  MoveL 627 to (56, 272.86, 210) mm, rotated rx -72.12 ry -13.76 rz 133.16 deg; joints [-11.184, -48.256, 111.238, -158.714, 116.997, -159.582, -1249.582]
  MoveL 628 to (57.57, 267.12, 200) mm, rotated rx -73 ry -11.66 rz 121.38 deg; joints [-11.86, -51.281, 112.071, -161.907, 109.412, -163.121, -1243.4]
  MoveL 629 to (58.59, 260.98, 190) mm, rotated rx -71.71 ry -12.29 rz 118.09 deg; joints [-12.413, -49.73, 111.982, -161.392, 113.738, -160.153, -1237.009]
  MoveL 630 to (58.95, 254.55, 180) mm, rotated rx -70.55 ry -13.02 rz 114.47 deg; joints [-12.913, -48.175, 111.692, -160.589, 117.696, -157.241, -1230.447]
  MoveL 631 to (58.59, 247.92, 170) mm, rotated rx -71.88 ry -10.84 rz 101.84 deg; joints [-13.52, -51.449, 112.574, -163.918, 109.603, -161.344, -1223.752]
  MoveL 632 to (57.45, 241.22, 160) mm, rotated rx -70.86 ry -11.6 rz 97.82 deg; joints [-13.978, -50.056, 112.473, -163.221, 113.479, -158.849, -1216.959]
  MoveL 633 to (55.51, 234.59, 150) mm, rotated rx -69.95 ry -12.44 rz 93.68 deg; joints [-14.39, -48.623, 112.206, -162.264, 117.149, -156.334, -1210.107]
  MoveL 634 to (52.77, 228.15, 140) mm, rotated rx -71.59 ry -10.32 rz 80.79 deg; joints [-14.925, -51.956, 113.016, -165.486, 108.844, -160.666, -1203.231]
  MoveL 635 to (49.26, 222.05, 130) mm, rotated rx -70.76 ry -11.22 rz 76.66 deg; joints [-15.304, -50.588, 112.931, -164.581, 112.697, -158.413, -1196.367]
  MoveL 636 to (45.04, 216.4, 120) mm, rotated rx -70.03 ry -12.23 rz 72.63 deg; joints [-15.637, -49.129, 112.673, -163.392, 116.478, -156.06, -1189.55]
  MoveL 637 to (40.19, 211.31, 110) mm, rotated rx -71.83 ry -10.32 rz 60.03 deg; joints [-16.092, -52.366, 113.385, -166.332, 108.333, -160.403, -1182.816]
  MoveL 638 to (34.83, 206.87, 100) mm, rotated rx -71.13 ry -11.44 rz 56.41 deg; joints [-16.388, -50.868, 113.282, -165.098, 112.545, -158.165, -1176.2]
  MoveL 639 to (29.06, 203.14, 90) mm, rotated rx -70.54 ry -12.69 rz 53.09 deg; joints [-16.632, -49.217, 112.963, -163.507, 116.784, -155.729, -1169.736]
  MoveL 640 to (23.03, 200.17, 80) mm, rotated rx -72.37 ry -11.13 rz 41.37 deg; joints [-17.001, -52.244, 113.649, -166.075, 109.258, -159.979, -1163.458]
  MoveL 641 to (16.86, 197.94, 70) mm, rotated rx -71.8 ry -12.55 rz 38.86 deg; joints [-17.193, -50.441, 113.427, -164.304, 114.153, -157.511, -1157.4]
  MoveL 642 to (10.69, 196.46, 60) mm, rotated rx -73.66 ry -11.39 rz 28.02 deg; joints [-17.464, -53.158, 113.849, -166.257, 107.044, -161.446, -1151.595]
  MoveL 643 to (4.64, 195.67, 50) mm, rotated rx -73.16 ry -13.02 rz 26.6 deg; joints [-17.59, -51.134, 113.679, -164.198, 112.728, -158.838, -1146.075]
  MoveL 644 to (-1.18, 195.49, 40) mm, rotated rx -72.85 ry -14.8 rz 25.84 deg; joints [-17.639, -48.817, 113.11, -161.546, 118.515, -155.811, -1140.872]
  MoveL 645 to (-6.67, 195.86, 30) mm, rotated rx -74.62 ry -14.16 rz 16.83 deg; joints [-17.801, -51.19, 113.743, -163.089, 112.896, -159.64, -1136.017]
  MoveL 646 to (-11.76, 196.67, 20) mm, rotated rx -76.4 ry -13.89 rz 8.51 deg; joints [-17.869, -53.24, 113.964, -163.907, 107.44, -163.077, -1131.54]
  MoveL 647 to (-16.38, 197.8, 10) mm, rotated rx -78.17 ry -13.98 rz 0.96 deg; joints [-17.851, -54.956, 113.848, -164.09, 102.301, -166.234, -1127.469]
  MoveL 648 to (-20.49, 199.16, 0) mm, rotated rx -78.17 ry -13.98 rz 0.96 deg; joints [-18.269, -54.883, 113.526, -164.417, 102.002, -166.09, -1127.469]
  Set speed (1000.0 mm/s)
  MoveL 649 to (-20.49, 199.16, 0) mm, rotated rx -78.17 ry -13.98 rz 0.96 deg; joints [-18.269, -54.883, 113.526, -164.417, 102.002, -166.09, -1127.469]
  Set speed (1000.0 mm/s)
  MoveL 650 to (37.11, 300.24, 290) mm, rotated rx -90 ry -25 rz 177.31 deg; joints [-2.318, -51.586, 102.108, -141.879, 96.357, -189.349, -1307.315]
  MoveL 651 to (37.11, 300.24, 290) mm, rotated rx -90 ry -25 rz -172.69 deg; joints [-2.265, -48.205, 103.066, -142.213, 108.813, -182.608, -1307.315]
  Set speed (60.0 mm/s)
  MoveL 652 to (43.85, 319.91, 290) mm, rotated rx -90 ry -25 rz -166.2 deg; joints [-2.265, -49.125, 102.977, -142.419, 108.014, -183.258, -1313.803]
  Set speed (1000.0 mm/s)
  MoveL 653 to (43.85, 319.91, 290) mm, rotated rx -90 ry -25 rz -166.2 deg; joints [-2.265, -49.125, 102.977, -142.419, 108.014, -183.258, -1313.803]
  Set speed (1000.0 mm/s)
  MoveL 654 to (-20.49, 199.16, 0) mm, rotated rx -90 ry -25 rz 31.39 deg; joints [-13.282, -51.572, 108.683, -149.29, 107.197, -175.931, -1151.385]
  MoveL 655 to (-20.49, 199.16, 0) mm, rotated rx -90 ry -25 rz 31.39 deg; joints [-13.282, -51.572, 108.683, -149.29, 107.197, -175.931, -1151.385]
  Set speed (60.0 mm/s)
  MoveL 656 to (-20.57, 178.36, 0) mm, rotated rx -90 ry -25 rz 45.86 deg; joints [-13.325, -48.191, 107.994, -147.492, 118.47, -169.661, -1155.856]
  Set speed (1000.0 mm/s)
  MoveL 657 to (-20.57, 178.36, 0) mm, rotated rx -90 ry -25 rz 45.86 deg; joints [-13.325, -48.191, 107.994, -147.492, 118.47, -169.661, -1155.856]
  Set speed (1000.0 mm/s)
  MoveL 658 to (-20.49, 199.16, 0) mm, rotated rx -90 ry -25 rz 31.39 deg; joints [-13.282, -51.572, 108.683, -149.29, 107.197, -175.931, -1151.385]
  MoveL 659 to (-20.49, 199.16, 0) mm, rotated rx -90 ry -25 rz 31.39 deg; joints [-13.282, -51.572, 108.683, -149.29, 107.197, -175.931, -1151.385]
  Set speed (60.0 mm/s)
  MoveL 660 to (-16.38, 197.8, 10) mm, rotated rx -90 ry -25 rz 35.25 deg; joints [-12.889, -51.522, 108.574, -149.026, 107.257, -176.155, -1155.247]
  MoveL 661 to (-11.76, 196.67, 20) mm, rotated rx -90 ry -25 rz 39.48 deg; joints [-12.496, -51.468, 108.459, -148.763, 107.315, -176.379, -1159.483]
  MoveL 662 to (-6.67, 195.86, 30) mm, rotated rx -90 ry -25 rz 44.06 deg; joints [-12.104, -51.409, 108.339, -148.502, 107.374, -176.604, -1164.062]
  MoveL 663 to (-1.18, 195.49, 40) mm, rotated rx -90 ry -25 rz 48.95 deg; joints [-11.713, -51.345, 108.212, -148.241, 107.432, -176.829, -1168.952]
  MoveL 664 to (4.64, 195.67, 50) mm, rotated rx -90 ry -25 rz 54.12 deg; joints [-11.323, -51.276, 108.079, -147.982, 107.491, -177.054, -1174.124]
  MoveL 665 to (10.69, 196.46, 60) mm, rotated rx -90 ry -25 rz 59.55 deg; joints [-10.933, -51.201, 107.94, -147.724, 107.551, -177.279, -1179.549]
  MoveL 666 to (16.86, 197.94, 70) mm, rotated rx -90 ry -25 rz 65.2 deg; joints [-10.544, -51.119, 107.796, -147.467, 107.612, -177.504, -1185.201]
  MoveL 667 to (23.03, 200.17, 80) mm, rotated rx -90 ry -25 rz 71.05 deg; joints [-10.156, -51.031, 107.645, -147.21, 107.675, -177.728, -1191.051]
  MoveL 668 to (29.06, 203.14, 90) mm, rotated rx -90 ry -25 rz 77.07 deg; joints [-9.769, -50.937, 107.489, -146.955, 107.738, -177.951, -1197.074]
  MoveL 669 to (34.83, 206.87, 100) mm, rotated rx -90 ry -25 rz 83.24 deg; joints [-9.383, -50.836, 107.326, -146.701, 107.803, -178.174, -1203.245]
  MoveL 670 to (40.19, 211.31, 110) mm, rotated rx -90 ry -25 rz 89.54 deg; joints [-8.998, -50.729, 107.158, -146.448, 107.869, -178.396, -1209.537]
  MoveL 671 to (45.04, 216.4, 120) mm, rotated rx -90 ry -25 rz 95.93 deg; joints [-8.614, -50.616, 106.984, -146.196, 107.936, -178.617, -1215.926]
  MoveL 672 to (49.26, 222.05, 130) mm, rotated rx -90 ry -25 rz 102.38 deg; joints [-8.231, -50.497, 106.804, -145.946, 108.004, -178.839, -1222.384]
  MoveL 673 to (52.77, 228.15, 140) mm, rotated rx -90 ry -25 rz 108.88 deg; joints [-7.849, -50.373, 106.617, -145.697, 108.072, -179.06, -1228.885]
  MoveL 674 to (55.51, 234.59, 150) mm, rotated rx -90 ry -25 rz 115.4 deg; joints [-7.468, -50.244, 106.425, -145.449, 108.139, -179.281, -1235.4]
  MoveL 675 to (57.45, 241.22, 160) mm, rotated rx -90 ry -25 rz 121.9 deg; joints [-7.088, -50.111, 106.226, -145.203, 108.206, -179.504, -1241.898]
  MoveL 676 to (58.59, 247.92, 170) mm, rotated rx -90 ry -25 rz 128.35 deg; joints [-6.709, -49.974, 106.022, -144.958, 108.271, -179.727, -1248.348]
  MoveL 677 to (58.95, 254.55, 180) mm, rotated rx -90 ry -25 rz 134.71 deg; joints [-6.332, -49.834, 105.811, -144.716, 108.334, -179.952, -1254.714]
  MoveL 678 to (58.59, 260.98, 190) mm, rotated rx -90 ry -25 rz 140.96 deg; joints [-5.956, -49.691, 105.593, -144.476, 108.396, -180.178, -1260.96]
  MoveL 679 to (57.57, 267.12, 200) mm, rotated rx -90 ry -25 rz 147.05 deg; joints [-5.581, -49.547, 105.37, -144.238, 108.454, -180.407, -1267.046]
  MoveL 680 to (56, 272.86, 210) mm, rotated rx -90 ry -25 rz 152.93 deg; joints [-5.207, -49.401, 105.139, -144.002, 108.509, -180.639, -1272.931]
  MoveL 681 to (53.98, 278.14, 220) mm, rotated rx -90 ry -25 rz 158.57 deg; joints [-4.834, -49.254, 104.903, -143.769, 108.56, -180.873, -1278.571]
  MoveL 682 to (51.62, 282.9, 230) mm, rotated rx -90 ry -25 rz 163.92 deg; joints [-4.463, -49.106, 104.66, -143.538, 108.608, -181.111, -1283.922]
  MoveL 683 to (49.06, 287.12, 240) mm, rotated rx -90 ry -25 rz 168.94 deg; joints [-4.093, -48.957, 104.41, -143.31, 108.652, -181.352, -1288.935]
  MoveL 684 to (46.4, 290.79, 250) mm, rotated rx -90 ry -25 rz 173.57 deg; joints [-3.725, -48.808, 104.155, -143.085, 108.692, -181.596, -1293.565]
  MoveL 685 to (43.78, 293.91, 260) mm, rotated rx -90 ry -25 rz 177.77 deg; joints [-3.358, -48.659, 103.892, -142.863, 108.728, -181.844, -1297.765]
  MoveL 686 to (41.29, 296.51, 270) mm, rotated rx -90 ry -25 rz -178.51 deg; joints [-2.992, -48.508, 103.623, -142.644, 108.76, -182.095, -1301.487]
  MoveL 687 to (39.03, 298.61, 280) mm, rotated rx -90 ry -25 rz -175.31 deg; joints [-2.628, -48.357, 103.348, -142.427, 108.788, -182.35, -1304.686]
  MoveL 688 to (37.11, 300.24, 290) mm, rotated rx -90 ry -25 rz -172.69 deg; joints [-2.265, -48.205, 103.066, -142.213, 108.813, -182.608, -1307.315]
  Set speed (1000.0 mm/s)
  MoveL 689 to (37.11, 300.24, 290) mm, rotated rx -90 ry -25 rz -172.69 deg; joints [-2.265, -48.205, 103.066, -142.213, 108.813, -182.608, -1307.315]
  Set speed (1000.0 mm/s)
  MoveL 690 to (43.85, 319.91, 290) mm, rotated rx -90 ry -25 rz -166.2 deg; joints [-2.265, -49.125, 102.977, -142.419, 108.014, -183.258, -1313.803]
  MoveL 691 to (43.85, 319.91, 290) mm, rotated rx -90 ry -25 rz -166.2 deg; joints [-2.265, -49.125, 102.977, -142.419, 108.014, -183.258, -1313.803]
  Set speed (60.0 mm/s)
  MoveL 692 to (46.6, 317.98, 280) mm, rotated rx -90 ry -25 rz -168.79 deg; joints [-2.628, -49.278, 103.258, -142.631, 107.986, -182.998, -1311.207]
  MoveL 693 to (49.86, 315.46, 270) mm, rotated rx -90 ry -25 rz -171.95 deg; joints [-2.992, -49.431, 103.534, -142.847, 107.954, -182.741, -1308.046]
  MoveL 694 to (53.49, 312.31, 260) mm, rotated rx -90 ry -25 rz -175.64 deg; joints [-3.358, -49.582, 103.802, -143.065, 107.919, -182.487, -1304.36]
  MoveL 695 to (57.36, 308.47, 250) mm, rotated rx -90 ry -25 rz -179.81 deg; joints [-3.725, -49.733, 104.064, -143.286, 107.88, -182.237, -1300.194]
  MoveL 696 to (61.34, 303.9, 240) mm, rotated rx -90 ry -25 rz 175.59 deg; joints [-4.093, -49.883, 104.32, -143.51, 107.836, -181.989, -1295.591]
  MoveL 697 to (65.27, 298.59, 230) mm, rotated rx -90 ry -25 rz 170.6 deg; joints [-4.463, -50.032, 104.569, -143.736, 107.789, -181.746, -1290.596]
  MoveL 698 to (68.98, 292.54, 220) mm, rotated rx -90 ry -25 rz 165.25 deg; joints [-4.834, -50.18, 104.811, -143.966, 107.738, -181.505, -1285.253]
  MoveL 699 to (72.31, 285.76, 210) mm, rotated rx -90 ry -25 rz 159.61 deg; joints [-5.207, -50.328, 105.047, -144.197, 107.683, -181.268, -1279.605]
  MoveL 700 to (75.1, 278.3, 200) mm, rotated rx -90 ry -25 rz 153.7 deg; joints [-5.581, -50.475, 105.276, -144.432, 107.624, -181.034, -1273.697]
  MoveL 701 to (77.2, 270.26, 190) mm, rotated rx -90 ry -25 rz 147.57 deg; joints [-5.956, -50.621, 105.499, -144.668, 107.562, -180.802, -1267.571]
  MoveL 702 to (78.47, 261.74, 180) mm, rotated rx -90 ry -25 rz 141.27 deg; joints [-6.332, -50.765, 105.715, -144.907, 107.496, -180.573, -1261.269]
  MoveL 703 to (78.79, 252.87, 170) mm, rotated rx -90 ry -25 rz 134.83 deg; joints [-6.709, -50.906, 105.925, -145.148, 107.428, -180.346, -1254.829]
  MoveL 704 to (78.09, 243.82, 160) mm, rotated rx -90 ry -25 rz 128.29 deg; joints [-7.088, -51.045, 106.129, -145.391, 107.357, -180.121, -1248.29]
  MoveL 705 to (76.31, 234.75, 150) mm, rotated rx -90 ry -25 rz 121.69 deg; joints [-7.468, -51.181, 106.326, -145.636, 107.285, -179.896, -1241.689]
  MoveL 706 to (73.44, 225.85, 140) mm, rotated rx -90 ry -25 rz 115.06 deg; joints [-7.849, -51.313, 106.518, -145.882, 107.212, -179.673, -1235.058]
  MoveL 707 to (69.5, 217.29, 130) mm, rotated rx -90 ry -25 rz 108.43 deg; joints [-8.231, -51.44, 106.703, -146.13, 107.138, -179.45, -1228.432]
  MoveL 708 to (64.57, 209.26, 120) mm, rotated rx -90 ry -25 rz 101.84 deg; joints [-8.614, -51.562, 106.882, -146.38, 107.064, -179.227, -1221.84]
  MoveL 709 to (58.74, 201.9, 110) mm, rotated rx -90 ry -25 rz 95.31 deg; joints [-8.998, -51.679, 107.055, -146.63, 106.991, -179.004, -1215.313]
  MoveL 710 to (52.14, 195.34, 100) mm, rotated rx -90 ry -25 rz 88.88 deg; joints [-9.383, -51.79, 107.223, -146.882, 106.918, -178.781, -1208.879]
  MoveL 711 to (44.91, 189.68, 90) mm, rotated rx -90 ry -25 rz 92.57 deg; joints [-9.833, -47.57, 106.798, -145.465, 118.969, -171.706, -1202.567]
  MoveL 712 to (37.24, 184.98, 80) mm, rotated rx -90 ry -25 rz 86.4 deg; joints [-10.217, -47.663, 106.955, -145.686, 118.911, -171.479, -1196.403]
  MoveL 713 to (29.3, 181.28, 70) mm, rotated rx -90 ry -25 rz 80.42 deg; joints [-10.603, -47.75, 107.107, -145.908, 118.855, -171.251, -1190.416]
  MoveL 714 to (21.27, 178.55, 60) mm, rotated rx -90 ry -25 rz 74.63 deg; joints [-10.989, -47.83, 107.252, -146.131, 118.799, -171.024, -1184.633]
  MoveL 715 to (13.31, 176.76, 50) mm, rotated rx -90 ry -25 rz 69.08 deg; joints [-11.377, -47.903, 107.391, -146.354, 118.744, -170.796, -1179.083]
  MoveL 716 to (5.58, 175.83, 40) mm, rotated rx -90 ry -25 rz 63.79 deg; joints [-11.765, -47.971, 107.524, -146.579, 118.689, -170.567, -1173.794]
  MoveL 717 to (-1.77, 175.65, 30) mm, rotated rx -90 ry -25 rz 58.8 deg; joints [-12.154, -48.034, 107.651, -146.805, 118.635, -170.34, -1168.796]
  MoveL 718 to (-8.64, 176.1, 20) mm, rotated rx -90 ry -25 rz 54.12 deg; joints [-12.543, -48.091, 107.771, -147.033, 118.58, -170.112, -1164.119]
  MoveL 719 to (-14.93, 177.06, 10) mm, rotated rx -90 ry -25 rz 49.79 deg; joints [-12.934, -48.143, 107.885, -147.261, 118.526, -169.886, -1159.795]
  MoveL 720 to (-20.57, 178.36, 0) mm, rotated rx -90 ry -25 rz 45.86 deg; joints [-13.325, -48.191, 107.994, -147.492, 118.47, -169.661, -1155.856]
  Set speed (1000.0 mm/s)
  MoveL 721 to (-20.57, 178.36, 0) mm, rotated rx -90 ry -25 rz 45.86 deg; joints [-13.325, -48.191, 107.994, -147.492, 118.47, -169.661, -1155.856]
  Set speed (1000.0 mm/s)
  MoveL 722 to (43.85, 319.91, 290) mm, rotated rx -90 ry -25 rz -166.2 deg; joints [-2.265, -49.125, 102.977, -142.419, 108.014, -183.258, -1313.803]
  MoveL 723 to (43.85, 319.91, 290) mm, rotated rx -90 ry -25 rz -166.2 deg; joints [-2.265, -49.125, 102.977, -142.419, 108.014, -183.258, -1313.803]
  Set speed (60.0 mm/s)
  MoveL 724 to (28.22, 306.19, 290) mm, rotated rx -90 ry -25 rz -161.42 deg; joints [-2.265, -48.176, 103.068, -142.207, 108.838, -182.588, -1318.582]
  Set speed (1000.0 mm/s)
  MoveL 725 to (28.22, 306.19, 290) mm, rotated rx -90 ry -25 rz -161.42 deg; joints [-2.265, -48.176, 103.068, -142.207, 108.838, -182.588, -1318.582]
  Set speed (1000.0 mm/s)
  MoveL 726 to (-20.57, 178.36, 0) mm, rotated rx -90 ry -25 rz 45.86 deg; joints [-13.325, -48.191, 107.994, -147.492, 118.47, -169.661, -1155.856]
  MoveL 727 to (-20.57, 178.36, 0) mm, rotated rx -90 ry -25 rz 45.86 deg; joints [-13.325, -48.191, 107.994, -147.492, 118.47, -169.661, -1155.856]
  Set speed (60.0 mm/s)
  MoveL 728 to (-10.16, 196.36, 0) mm, rotated rx -90 ry -25 rz 40.93 deg; joints [-13.282, -51.585, 108.681, -149.292, 107.186, -175.938, -1160.929]
  Set speed (1000.0 mm/s)
  MoveL 729 to (-10.16, 196.36, 0) mm, rotated rx -90 ry -25 rz 40.93 deg; joints [-13.282, -51.585, 108.681, -149.292, 107.186, -175.938, -1160.929]
  Set speed (1000.0 mm/s)
  MoveL 730 to (-20.57, 178.36, 0) mm, rotated rx -90 ry -25 rz 45.86 deg; joints [-13.325, -48.191, 107.994, -147.492, 118.47, -169.661, -1155.856]
  MoveL 731 to (-20.57, 178.36, 0) mm, rotated rx -90 ry -25 rz 45.86 deg; joints [-13.325, -48.191, 107.994, -147.492, 118.47, -169.661, -1155.856]
  Set speed (60.0 mm/s)
  MoveL 732 to (-14.93, 177.06, 10) mm, rotated rx -90 ry -25 rz 49.79 deg; joints [-12.934, -48.143, 107.885, -147.261, 118.526, -169.886, -1159.795]
  MoveL 733 to (-8.64, 176.1, 20) mm, rotated rx -90 ry -25 rz 54.12 deg; joints [-12.543, -48.091, 107.771, -147.033, 118.58, -170.112, -1164.119]
  MoveL 734 to (-1.77, 175.65, 30) mm, rotated rx -90 ry -25 rz 58.8 deg; joints [-12.154, -48.034, 107.651, -146.805, 118.635, -170.34, -1168.796]
  MoveL 735 to (5.58, 175.83, 40) mm, rotated rx -90 ry -25 rz 63.79 deg; joints [-11.765, -47.971, 107.524, -146.579, 118.689, -170.567, -1173.794]
  MoveL 736 to (13.31, 176.76, 50) mm, rotated rx -90 ry -25 rz 69.08 deg; joints [-11.377, -47.903, 107.391, -146.354, 118.744, -170.796, -1179.083]
  MoveL 737 to (21.27, 178.55, 60) mm, rotated rx -90 ry -25 rz 74.63 deg; joints [-10.989, -47.83, 107.252, -146.131, 118.799, -171.024, -1184.633]
  MoveL 738 to (29.3, 181.28, 70) mm, rotated rx -90 ry -25 rz 80.42 deg; joints [-10.603, -47.75, 107.107, -145.908, 118.855, -171.251, -1190.416]
  MoveL 739 to (37.24, 184.98, 80) mm, rotated rx -90 ry -25 rz 86.4 deg; joints [-10.217, -47.663, 106.955, -145.686, 118.911, -171.479, -1196.403]
  MoveL 740 to (44.91, 189.68, 90) mm, rotated rx -90 ry -25 rz 92.57 deg; joints [-9.833, -47.57, 106.798, -145.465, 118.969, -171.706, -1202.567]
  MoveL 741 to (52.14, 195.34, 100) mm, rotated rx -90 ry -25 rz 88.88 deg; joints [-9.383, -51.79, 107.223, -146.882, 106.918, -178.781, -1208.879]
  MoveL 742 to (58.74, 201.9, 110) mm, rotated rx -90 ry -25 rz 95.31 deg; joints [-8.998, -51.679, 107.055, -146.63, 106.991, -179.004, -1215.313]
  MoveL 743 to (64.57, 209.26, 120) mm, rotated rx -90 ry -25 rz 101.84 deg; joints [-8.614, -51.562, 106.882, -146.38, 107.064, -179.227, -1221.84]
  MoveL 744 to (69.5, 217.29, 130) mm, rotated rx -90 ry -25 rz 108.43 deg; joints [-8.231, -51.44, 106.703, -146.13, 107.138, -179.45, -1228.432]
  MoveL 745 to (73.44, 225.85, 140) mm, rotated rx -90 ry -25 rz 115.06 deg; joints [-7.849, -51.313, 106.518, -145.882, 107.212, -179.673, -1235.058]
  MoveL 746 to (76.31, 234.75, 150) mm, rotated rx -90 ry -25 rz 121.69 deg; joints [-7.468, -51.181, 106.326, -145.636, 107.285, -179.896, -1241.689]
  MoveL 747 to (78.09, 243.82, 160) mm, rotated rx -90 ry -25 rz 128.29 deg; joints [-7.088, -51.045, 106.129, -145.391, 107.357, -180.121, -1248.29]
  MoveL 748 to (78.79, 252.87, 170) mm, rotated rx -90 ry -25 rz 134.83 deg; joints [-6.709, -50.906, 105.925, -145.148, 107.428, -180.346, -1254.829]
  MoveL 749 to (78.47, 261.74, 180) mm, rotated rx -90 ry -25 rz 141.27 deg; joints [-6.332, -50.765, 105.715, -144.907, 107.496, -180.573, -1261.269]
  MoveL 750 to (77.2, 270.26, 190) mm, rotated rx -90 ry -25 rz 147.57 deg; joints [-5.956, -50.621, 105.499, -144.668, 107.562, -180.802, -1267.571]
  MoveL 751 to (75.1, 278.3, 200) mm, rotated rx -90 ry -25 rz 153.7 deg; joints [-5.581, -50.475, 105.276, -144.432, 107.624, -181.034, -1273.697]
  MoveL 752 to (72.31, 285.76, 210) mm, rotated rx -90 ry -25 rz 159.61 deg; joints [-5.207, -50.328, 105.047, -144.197, 107.683, -181.268, -1279.605]
  MoveL 753 to (68.98, 292.54, 220) mm, rotated rx -90 ry -25 rz 165.25 deg; joints [-4.834, -50.18, 104.811, -143.966, 107.738, -181.505, -1285.253]
  MoveL 754 to (65.27, 298.59, 230) mm, rotated rx -90 ry -25 rz 170.6 deg; joints [-4.463, -50.032, 104.569, -143.736, 107.789, -181.746, -1290.596]
  MoveL 755 to (61.34, 303.9, 240) mm, rotated rx -90 ry -25 rz 175.59 deg; joints [-4.093, -49.883, 104.32, -143.51, 107.836, -181.989, -1295.591]
  MoveL 756 to (57.36, 308.47, 250) mm, rotated rx -90 ry -25 rz -179.81 deg; joints [-3.725, -49.733, 104.064, -143.286, 107.88, -182.237, -1300.194]
  MoveL 757 to (53.49, 312.31, 260) mm, rotated rx -90 ry -25 rz -175.64 deg; joints [-3.358, -49.582, 103.802, -143.065, 107.919, -182.487, -1304.36]
  MoveL 758 to (49.86, 315.46, 270) mm, rotated rx -90 ry -25 rz -171.95 deg; joints [-2.992, -49.431, 103.534, -142.847, 107.954, -182.741, -1308.046]
  MoveL 759 to (46.6, 317.98, 280) mm, rotated rx -90 ry -25 rz -168.79 deg; joints [-2.628, -49.278, 103.258, -142.631, 107.986, -182.998, -1311.207]
  MoveL 760 to (43.85, 319.91, 290) mm, rotated rx -90 ry -25 rz -166.2 deg; joints [-2.265, -49.125, 102.977, -142.419, 108.014, -183.258, -1313.803]
  Set speed (1000.0 mm/s)
  MoveL 761 to (43.85, 319.91, 290) mm, rotated rx -90 ry -25 rz -166.2 deg; joints [-2.265, -49.125, 102.977, -142.419, 108.014, -183.258, -1313.803]
  Set speed (1000.0 mm/s)
  MoveL 762 to (28.22, 306.19, 290) mm, rotated rx -90 ry -25 rz -161.42 deg; joints [-2.265, -48.176, 103.068, -142.207, 108.838, -182.588, -1318.582]
  MoveL 763 to (28.22, 306.19, 290) mm, rotated rx -90 ry -25 rz -161.42 deg; joints [-2.265, -48.176, 103.068, -142.207, 108.838, -182.588, -1318.582]
  Set speed (60.0 mm/s)
  MoveL 764 to (30.4, 304.94, 280) mm, rotated rx -90 ry -25 rz -164.08 deg; joints [-2.628, -48.326, 103.35, -142.42, 108.814, -182.329, -1315.919]
  MoveL 765 to (33, 303.28, 270) mm, rotated rx -90 ry -25 rz -167.32 deg; joints [-2.992, -48.475, 103.626, -142.636, 108.788, -182.073, -1312.679]
  MoveL 766 to (35.92, 301.18, 260) mm, rotated rx -90 ry -25 rz -171.09 deg; joints [-3.358, -48.623, 103.895, -142.855, 108.758, -181.82, -1308.905]
  MoveL 767 to (39.07, 298.58, 250) mm, rotated rx -90 ry -25 rz -175.36 deg; joints [-3.725, -48.771, 104.158, -143.077, 108.724, -181.57, -1304.643]
  MoveL 768 to (42.34, 295.45, 240) mm, rotated rx -90 ry -25 rz 179.94 deg; joints [-4.093, -48.917, 104.414, -143.302, 108.687, -181.325, -1299.941]
  MoveL 769 to (45.62, 291.76, 230) mm, rotated rx -90 ry -25 rz 174.85 deg; joints [-4.463, -49.064, 104.663, -143.529, 108.645, -181.082, -1294.846]
  MoveL 770 to (48.8, 287.5, 220) mm, rotated rx -90 ry -25 rz 169.41 deg; joints [-4.834, -49.209, 104.907, -143.759, 108.599, -180.843, -1289.406]
  MoveL 771 to (51.74, 282.68, 210) mm, rotated rx -90 ry -25 rz 163.67 deg; joints [-5.207, -49.355, 105.143, -143.992, 108.55, -180.608, -1283.668]
  MoveL 772 to (54.33, 277.32, 200) mm, rotated rx -90 ry -25 rz 157.68 deg; joints [-5.581, -49.499, 105.373, -144.227, 108.496, -180.375, -1277.679]
  MoveL 773 to (56.44, 271.47, 190) mm, rotated rx -90 ry -25 rz 151.49 deg; joints [-5.956, -49.643, 105.597, -144.465, 108.439, -180.146, -1271.486]
  MoveL 774 to (57.96, 265.2, 180) mm, rotated rx -90 ry -25 rz 145.13 deg; joints [-6.332, -49.785, 105.815, -144.706, 108.378, -179.919, -1265.13]
  MoveL 775 to (58.8, 258.62, 170) mm, rotated rx -90 ry -25 rz 138.66 deg; joints [-6.709, -49.925, 106.026, -144.948, 108.315, -179.695, -1258.655]
  MoveL 776 to (58.89, 251.83, 160) mm, rotated rx -90 ry -25 rz 132.1 deg; joints [-7.088, -50.063, 106.23, -145.193, 108.249, -179.472, -1252.098]
  MoveL 777 to (58.18, 244.95, 150) mm, rotated rx -90 ry -25 rz 125.5 deg; joints [-7.468, -50.197, 106.429, -145.439, 108.181, -179.251, -1245.497]
  MoveL 778 to (56.65, 238.12, 140) mm, rotated rx -90 ry -25 rz 118.89 deg; joints [-7.849, -50.329, 106.621, -145.688, 108.112, -179.031, -1238.886]
  MoveL 779 to (54.3, 231.49, 130) mm, rotated rx -90 ry -25 rz 112.3 deg; joints [-8.231, -50.455, 106.807, -145.937, 108.042, -178.812, -1232.295]
  MoveL 780 to (51.17, 225.17, 120) mm, rotated rx -90 ry -25 rz 105.76 deg; joints [-8.614, -50.578, 106.987, -146.189, 107.971, -178.593, -1225.756]
  MoveL 781 to (47.33, 219.29, 110) mm, rotated rx -90 ry -25 rz 99.3 deg; joints [-8.998, -50.694, 107.161, -146.441, 107.901, -178.374, -1219.296]
  MoveL 782 to (42.85, 213.95, 100) mm, rotated rx -90 ry -25 rz 92.94 deg; joints [-9.383, -50.806, 107.329, -146.695, 107.831, -178.154, -1212.941]
  MoveL 783 to (37.86, 209.24, 90) mm, rotated rx -90 ry -25 rz 86.72 deg; joints [-9.769, -50.911, 107.491, -146.95, 107.762, -177.935, -1206.718]
  MoveL 784 to (32.46, 205.23, 80) mm, rotated rx -90 ry -25 rz 80.65 deg; joints [-10.156, -51.009, 107.647, -147.206, 107.695, -177.714, -1200.653]
  MoveL 785 to (26.8, 201.92, 70) mm, rotated rx -90 ry -25 rz 74.77 deg; joints [-10.544, -51.102, 107.797, -147.463, 107.628, -177.493, -1194.769]
  MoveL 786 to (21, 199.35, 60) mm, rotated rx -90 ry -25 rz 69.09 deg; joints [-10.933, -51.188, 107.942, -147.721, 107.563, -177.272, -1189.094]
  MoveL 787 to (15.19, 197.47, 50) mm, rotated rx -90 ry -25 rz 63.65 deg; joints [-11.323, -51.268, 108.08, -147.981, 107.498, -177.05, -1183.653]
  MoveL 788 to (9.5, 196.25, 40) mm, rotated rx -90 ry -25 rz 58.47 deg; joints [-11.713, -51.342, 108.212, -148.241, 107.435, -176.827, -1178.473]
  MoveL 789 to (4.03, 195.62, 30) mm, rotated rx -90 ry -25 rz 53.58 deg; joints [-12.104, -51.41, 108.339, -148.502, 107.373, -176.605, -1173.581]
  MoveL 790 to (-1.12, 195.49, 20) mm, rotated rx -90 ry -25 rz 49.01 deg; joints [-12.496, -51.473, 108.459, -148.764, 107.31, -176.382, -1169.007]
  MoveL 791 to (-5.87, 195.78, 10) mm, rotated rx -90 ry -25 rz 44.78 deg; joints [-12.889, -51.531, 108.573, -149.027, 107.248, -176.16, -1164.779]
  MoveL 792 to (-10.16, 196.36, 0) mm, rotated rx -90 ry -25 rz 40.93 deg; joints [-13.282, -51.585, 108.681, -149.292, 107.186, -175.938, -1160.929]
  Set speed (1000.0 mm/s)
  MoveL 793 to (-10.16, 196.36, 0) mm, rotated rx -90 ry -25 rz 40.93 deg; joints [-13.282, -51.585, 108.681, -149.292, 107.186, -175.938, -1160.929]
  Set speed (1000.0 mm/s)
  MoveL 794 to (28.22, 306.19, 290) mm, rotated rx -90 ry -25 rz -161.42 deg; joints [-2.265, -48.176, 103.068, -142.207, 108.838, -182.588, -1318.582]
  MoveL 795 to (28.22, 306.19, 290) mm, rotated rx -90 ry -25 rz -161.42 deg; joints [-2.265, -48.176, 103.068, -142.207, 108.838, -182.588, -1318.582]
  Set speed (60.0 mm/s)
  MoveL 796 to (-21.11, 309.47, 290) mm, rotated rx -90 ry -25 rz -106.89 deg; joints [-2.265, -48.16, 103.069, -142.203, 108.851, -182.577, -1373.11]
  Set speed (1000.0 mm/s)
  MoveL 797 to (-21.11, 309.47, 290) mm, rotated rx -90 ry -25 rz -106.89 deg; joints [-2.265, -48.16, 103.069, -142.203, 108.851, -182.577, -1373.11]
  Set speed (1000.0 mm/s)
  MoveL 798 to (-10.16, 196.36, 0) mm, rotated rx -90 ry -25 rz 40.93 deg; joints [-13.282, -51.585, 108.681, -149.292, 107.186, -175.938, -1520.929]
  MoveL 799 to (-10.16, 196.36, 0) mm, rotated rx -90 ry -25 rz 40.93 deg; joints [-13.282, -51.585, 108.681, -149.292, 107.186, -175.938, -1520.929]
  Set speed (60.0 mm/s)
  MoveL 800 to (37.62, 209.05, 0) mm, rotated rx -90 ry -25 rz 86.44 deg; joints [-13.282, -51.529, 108.687, -149.283, 107.238, -175.906, -1566.442]
  Set speed (1000.0 mm/s)
  MoveL 801 to (37.62, 209.05, 0) mm, rotated rx -90 ry -25 rz 86.44 deg; joints [-13.282, -51.529, 108.687, -149.283, 107.238, -175.906, -1566.442]
  Set speed (1000.0 mm/s)
  MoveL 802 to (-10.16, 196.36, 0) mm, rotated rx -90 ry -25 rz 40.93 deg; joints [-13.282, -51.585, 108.681, -149.292, 107.186, -175.938, -1520.929]
  MoveL 803 to (-10.16, 196.36, 0) mm, rotated rx -90 ry -25 rz 40.93 deg; joints [-13.282, -51.585, 108.681, -149.292, 107.186, -175.938, -1520.929]
  Set speed (60.0 mm/s)
  MoveL 804 to (-5.87, 195.78, 10) mm, rotated rx -90 ry -25 rz 44.78 deg; joints [-12.889, -51.531, 108.573, -149.027, 107.248, -176.16, -1524.779]
  MoveL 805 to (-1.12, 195.49, 20) mm, rotated rx -90 ry -25 rz 49.01 deg; joints [-12.496, -51.473, 108.459, -148.764, 107.31, -176.382, -1529.007]
  MoveL 806 to (4.03, 195.62, 30) mm, rotated rx -90 ry -25 rz 53.58 deg; joints [-12.104, -51.41, 108.339, -148.502, 107.373, -176.605, -1533.581]
  MoveL 807 to (9.5, 196.25, 40) mm, rotated rx -90 ry -25 rz 58.47 deg; joints [-11.713, -51.342, 108.212, -148.241, 107.435, -176.827, -1538.473]
  MoveL 808 to (15.19, 197.47, 50) mm, rotated rx -90 ry -25 rz 63.65 deg; joints [-11.323, -51.268, 108.08, -147.981, 107.498, -177.05, -1543.653]
  MoveL 809 to (21, 199.35, 60) mm, rotated rx -90 ry -25 rz 69.09 deg; joints [-10.933, -51.188, 107.942, -147.721, 107.563, -177.272, -1549.094]
  MoveL 810 to (26.8, 201.92, 70) mm, rotated rx -90 ry -25 rz 74.77 deg; joints [-10.544, -51.102, 107.797, -147.463, 107.628, -177.493, -1554.769]
  MoveL 811 to (32.46, 205.23, 80) mm, rotated rx -90 ry -25 rz 80.65 deg; joints [-10.156, -51.009, 107.647, -147.206, 107.695, -177.714, -1560.653]
  MoveL 812 to (37.86, 209.24, 90) mm, rotated rx -90 ry -25 rz 86.72 deg; joints [-9.769, -50.911, 107.491, -146.95, 107.762, -177.935, -1566.718]
  MoveL 813 to (42.85, 213.95, 100) mm, rotated rx -90 ry -25 rz 92.94 deg; joints [-9.383, -50.806, 107.329, -146.695, 107.831, -178.154, -1572.941]
  MoveL 814 to (47.33, 219.29, 110) mm, rotated rx -90 ry -25 rz 99.3 deg; joints [-8.998, -50.694, 107.161, -146.441, 107.901, -178.374, -1579.296]
  MoveL 815 to (51.17, 225.17, 120) mm, rotated rx -90 ry -25 rz 105.76 deg; joints [-8.614, -50.578, 106.987, -146.189, 107.971, -178.593, -1585.756]
  MoveL 816 to (54.3, 231.49, 130) mm, rotated rx -90 ry -25 rz 112.3 deg; joints [-8.231, -50.455, 106.807, -145.937, 108.042, -178.812, -1592.295]
  MoveL 817 to (56.65, 238.12, 140) mm, rotated rx -90 ry -25 rz 118.89 deg; joints [-7.849, -50.329, 106.621, -145.688, 108.112, -179.031, -1598.886]
  MoveL 818 to (58.18, 244.95, 150) mm, rotated rx -90 ry -25 rz 125.5 deg; joints [-7.468, -50.197, 106.429, -145.439, 108.181, -179.251, -1605.497]
  MoveL 819 to (58.89, 251.83, 160) mm, rotated rx -90 ry -25 rz 132.1 deg; joints [-7.088, -50.063, 106.23, -145.193, 108.249, -179.472, -1612.098]
  MoveL 820 to (58.8, 258.62, 170) mm, rotated rx -90 ry -25 rz 138.66 deg; joints [-6.709, -49.925, 106.026, -144.948, 108.315, -179.695, -1618.655]
  MoveL 821 to (57.96, 265.2, 180) mm, rotated rx -90 ry -25 rz 145.13 deg; joints [-6.332, -49.785, 105.815, -144.706, 108.378, -179.919, -1625.13]
  MoveL 822 to (56.44, 271.47, 190) mm, rotated rx -90 ry -25 rz 151.49 deg; joints [-5.956, -49.643, 105.597, -144.465, 108.439, -180.146, -1631.486]
  MoveL 823 to (54.33, 277.32, 200) mm, rotated rx -90 ry -25 rz 157.68 deg; joints [-5.581, -49.499, 105.373, -144.227, 108.496, -180.375, -1637.679]
  MoveL 824 to (51.74, 282.68, 210) mm, rotated rx -90 ry -25 rz 163.67 deg; joints [-5.207, -49.355, 105.143, -143.992, 108.55, -180.608, -1643.668]
  MoveL 825 to (48.8, 287.5, 220) mm, rotated rx -90 ry -25 rz 169.41 deg; joints [-4.834, -49.209, 104.907, -143.759, 108.599, -180.843, -1649.406]
  MoveL 826 to (45.62, 291.76, 230) mm, rotated rx -90 ry -25 rz 174.85 deg; joints [-4.463, -49.064, 104.663, -143.529, 108.645, -181.082, -1654.846]
  MoveL 827 to (42.34, 295.45, 240) mm, rotated rx -90 ry -25 rz 179.94 deg; joints [-4.093, -48.917, 104.414, -143.302, 108.687, -181.325, -1659.941]
  MoveL 828 to (39.07, 298.58, 250) mm, rotated rx -90 ry -25 rz -175.36 deg; joints [-3.725, -48.771, 104.158, -143.077, 108.724, -181.57, -1664.643]
  MoveL 829 to (35.92, 301.18, 260) mm, rotated rx -90 ry -25 rz -171.09 deg; joints [-3.358, -48.623, 103.895, -142.855, 108.758, -181.82, -1668.905]
  MoveL 830 to (33, 303.28, 270) mm, rotated rx -90 ry -25 rz -167.32 deg; joints [-2.992, -48.475, 103.626, -142.636, 108.788, -182.073, -1672.679]
  MoveL 831 to (30.4, 304.94, 280) mm, rotated rx -90 ry -25 rz -164.08 deg; joints [-2.628, -48.326, 103.35, -142.42, 108.814, -182.329, -1675.919]
  MoveL 832 to (28.22, 306.19, 290) mm, rotated rx -90 ry -25 rz -161.42 deg; joints [-2.265, -48.176, 103.068, -142.207, 108.838, -182.588, -1678.582]
  Set speed (1000.0 mm/s)
  MoveL 833 to (28.22, 306.19, 290) mm, rotated rx -90 ry -25 rz -161.42 deg; joints [-2.265, -48.176, 103.068, -142.207, 108.838, -182.588, -1678.582]
  Set speed (1000.0 mm/s)
  MoveL 834 to (-21.11, 309.47, 290) mm, rotated rx -90 ry -25 rz -106.89 deg; joints [-2.265, -48.16, 103.069, -142.203, 108.851, -182.577, -1733.11]
  MoveL 835 to (-21.11, 309.47, 290) mm, rotated rx -90 ry -25 rz -106.89 deg; joints [-2.265, -48.16, 103.069, -142.203, 108.851, -182.577, -1733.11]
  Set speed (60.0 mm/s)
  MoveL 836 to (-18.74, 310.33, 280) mm, rotated rx -90 ry -25 rz -109.58 deg; joints [-2.628, -48.3, 103.352, -142.414, 108.837, -182.31, -1730.424]
  MoveL 837 to (-15.8, 311.23, 270) mm, rotated rx -90 ry -25 rz -112.86 deg; joints [-2.992, -48.436, 103.629, -142.628, 108.822, -182.046, -1727.138]
  MoveL 838 to (-12.3, 312.09, 260) mm, rotated rx -90 ry -25 rz -116.71 deg; joints [-3.358, -48.569, 103.899, -142.843, 108.804, -181.783, -1723.29]
  MoveL 839 to (-8.28, 312.8, 250) mm, rotated rx -90 ry -25 rz -121.08 deg; joints [-3.725, -48.7, 104.163, -143.062, 108.785, -181.522, -1718.917]
  MoveL 840 to (-3.78, 313.26, 240) mm, rotated rx -90 ry -25 rz -125.94 deg; joints [-4.093, -48.829, 104.421, -143.282, 108.763, -181.265, -1714.059]
  MoveL 841 to (1.16, 313.37, 230) mm, rotated rx -90 ry -25 rz -131.24 deg; joints [-4.463, -48.957, 104.672, -143.506, 108.737, -181.01, -1708.756]
  MoveL 842 to (6.46, 313.03, 220) mm, rotated rx -90 ry -25 rz -136.95 deg; joints [-4.834, -49.084, 104.916, -143.732, 108.709, -180.759, -1703.053]
  MoveL 843 to (12.04, 312.14, 210) mm, rotated rx -90 ry -25 rz -143.01 deg; joints [-5.207, -49.21, 105.155, -143.961, 108.676, -180.511, -1696.995]
  MoveL 844 to (17.8, 310.63, 200) mm, rotated rx -90 ry -25 rz -149.37 deg; joints [-5.581, -49.336, 105.386, -144.193, 108.639, -180.267, -1690.629]
  MoveL 845 to (23.62, 308.44, 190) mm, rotated rx -90 ry -25 rz -155.99 deg; joints [-5.956, -49.463, 105.612, -144.428, 108.597, -180.027, -1684.006]
  MoveL 846 to (29.38, 305.54, 180) mm, rotated rx -90 ry -25 rz -162.82 deg; joints [-6.332, -49.59, 105.83, -144.665, 108.55, -179.791, -1677.176]
  MoveL 847 to (34.94, 301.92, 170) mm, rotated rx -90 ry -25 rz -169.81 deg; joints [-6.709, -49.717, 106.043, -144.905, 108.498, -179.559, -1670.188]
  MoveL 848 to (40.17, 297.58, 160) mm, rotated rx -90 ry -25 rz -176.91 deg; joints [-7.088, -49.845, 106.248, -145.148, 108.442, -179.33, -1663.094]
  MoveL 849 to (44.94, 292.58, 150) mm, rotated rx -90 ry -25 rz 175.94 deg; joints [-7.468, -49.972, 106.447, -145.394, 108.381, -179.106, -1655.941]
  MoveL 850 to (49.15, 286.99, 140) mm, rotated rx -90 ry -25 rz 168.77 deg; joints [-7.849, -50.1, 106.64, -145.642, 108.316, -178.884, -1648.774]
  MoveL 851 to (52.68, 280.9, 130) mm, rotated rx -90 ry -25 rz 161.64 deg; joints [-8.231, -50.226, 106.827, -145.892, 108.247, -178.665, -1641.638]
  MoveL 852 to (55.46, 274.42, 120) mm, rotated rx -90 ry -25 rz 154.57 deg; joints [-8.614, -50.351, 107.007, -146.144, 108.175, -178.449, -1634.572]
  MoveL 853 to (57.44, 267.68, 110) mm, rotated rx -90 ry -25 rz 147.61 deg; joints [-8.998, -50.474, 107.18, -146.398, 108.101, -178.234, -1627.613]
  MoveL 854 to (58.6, 260.81, 100) mm, rotated rx -90 ry -25 rz 140.79 deg; joints [-9.383, -50.593, 107.348, -146.654, 108.024, -178.021, -1620.794]
  MoveL 855 to (58.95, 253.96, 90) mm, rotated rx -90 ry -25 rz 134.15 deg; joints [-9.769, -50.71, 107.509, -146.912, 107.945, -177.809, -1614.147]
  MoveL 856 to (58.51, 247.24, 80) mm, rotated rx -90 ry -25 rz 127.7 deg; joints [-10.156, -50.822, 107.664, -147.171, 107.866, -177.598, -1607.701]
  MoveL 857 to (57.35, 240.79, 70) mm, rotated rx -90 ry -25 rz 121.48 deg; joints [-10.544, -50.93, 107.813, -147.431, 107.786, -177.387, -1601.482]
  MoveL 858 to (55.55, 234.7, 60) mm, rotated rx -90 ry -25 rz 115.52 deg; joints [-10.933, -51.032, 107.956, -147.693, 107.706, -177.177, -1595.517]
  MoveL 859 to (53.21, 229.07, 50) mm, rotated rx -90 ry -25 rz 109.83 deg; joints [-11.323, -51.129, 108.092, -147.955, 107.627, -176.966, -1589.83]
  MoveL 860 to (50.45, 223.94, 40) mm, rotated rx -90 ry -25 rz 104.45 deg; joints [-11.713, -51.221, 108.223, -148.219, 107.548, -176.754, -1584.447]
  MoveL 861 to (47.39, 219.37, 30) mm, rotated rx -90 ry -25 rz 99.39 deg; joints [-12.104, -51.307, 108.348, -148.483, 107.469, -176.543, -1579.391]
  MoveL 862 to (44.15, 215.37, 20) mm, rotated rx -90 ry -25 rz 94.69 deg; joints [-12.496, -51.387, 108.467, -148.749, 107.391, -176.331, -1574.688]
  MoveL 863 to (40.85, 211.93, 10) mm, rotated rx -90 ry -25 rz 90.36 deg; joints [-12.889, -51.461, 108.58, -149.015, 107.314, -176.119, -1570.363]
  MoveL 864 to (37.62, 209.05, 0) mm, rotated rx -90 ry -25 rz 86.44 deg; joints [-13.282, -51.529, 108.687, -149.283, 107.238, -175.906, -1566.442]
  Set speed (1000.0 mm/s)
  MoveL 865 to (37.62, 209.05, 0) mm, rotated rx -90 ry -25 rz 86.44 deg; joints [-13.282, -51.529, 108.687, -149.283, 107.238, -175.906, -1566.442]
  Set speed (1000.0 mm/s)
  MoveL 866 to (-21.11, 309.47, 290) mm, rotated rx -90 ry -25 rz -106.89 deg; joints [-2.265, -48.16, 103.069, -142.203, 108.851, -182.577, -1733.11]
  MoveL 867 to (-21.11, 309.47, 290) mm, rotated rx -90 ry -25 rz -106.89 deg; joints [-2.265, -48.16, 103.069, -142.203, 108.851, -182.577, -1733.11]
  Set speed (60.0 mm/s)
  MoveL 868 to (-34.79, 325.15, 290) mm, rotated rx -90 ry -25 rz -101.9 deg; joints [-2.265, -49.106, 102.979, -142.415, 108.03, -183.245, -1738.101]
  Set speed (1000.0 mm/s)
  MoveL 869 to (-34.79, 325.15, 290) mm, rotated rx -90 ry -25 rz -101.9 deg; joints [-2.265, -49.106, 102.979, -142.415, 108.03, -183.245, -1738.101]
  Set speed (1000.0 mm/s)
  MoveL 870 to (37.62, 209.05, 0) mm, rotated rx -90 ry -25 rz 86.44 deg; joints [-13.282, -51.529, 108.687, -149.283, 107.238, -175.906, -1566.442]
  MoveL 871 to (37.62, 209.05, 0) mm, rotated rx -90 ry -25 rz 86.44 deg; joints [-13.282, -51.529, 108.687, -149.283, 107.238, -175.906, -1566.442]
  Set speed (60.0 mm/s)
  MoveL 872 to (55.59, 198.58, 0) mm, rotated rx -90 ry -25 rz 102.15 deg; joints [-13.325, -48.121, 107.993, -147.471, 118.529, -169.618, -1572.15]
  Set speed (1000.0 mm/s)
  MoveL 873 to (55.59, 198.58, 0) mm, rotated rx -90 ry -25 rz 102.15 deg; joints [-13.325, -48.121, 107.993, -147.471, 118.529, -169.618, -1572.15]
  Set speed (1000.0 mm/s)
  MoveL 874 to (37.62, 209.05, 0) mm, rotated rx -90 ry -25 rz 86.44 deg; joints [-13.282, -51.529, 108.687, -149.283, 107.238, -175.906, -1566.442]
  MoveL 875 to (37.62, 209.05, 0) mm, rotated rx -90 ry -25 rz 86.44 deg; joints [-13.282, -51.529, 108.687, -149.283, 107.238, -175.906, -1566.442]
  Set speed (60.0 mm/s)
  MoveL 876 to (40.85, 211.93, 10) mm, rotated rx -90 ry -25 rz 90.36 deg; joints [-12.889, -51.461, 108.58, -149.015, 107.314, -176.119, -1570.363]
  MoveL 877 to (44.15, 215.37, 20) mm, rotated rx -90 ry -25 rz 94.69 deg; joints [-12.496, -51.387, 108.467, -148.749, 107.391, -176.331, -1574.688]
  MoveL 878 to (47.39, 219.37, 30) mm, rotated rx -90 ry -25 rz 99.39 deg; joints [-12.104, -51.307, 108.348, -148.483, 107.469, -176.543, -1579.391]
  MoveL 879 to (50.45, 223.94, 40) mm, rotated rx -90 ry -25 rz 104.45 deg; joints [-11.713, -51.221, 108.223, -148.219, 107.548, -176.754, -1584.447]
  MoveL 880 to (53.21, 229.07, 50) mm, rotated rx -90 ry -25 rz 109.83 deg; joints [-11.323, -51.129, 108.092, -147.955, 107.627, -176.966, -1589.83]
  MoveL 881 to (55.55, 234.7, 60) mm, rotated rx -90 ry -25 rz 115.52 deg; joints [-10.933, -51.032, 107.956, -147.693, 107.706, -177.177, -1595.517]
  MoveL 882 to (57.35, 240.79, 70) mm, rotated rx -90 ry -25 rz 121.48 deg; joints [-10.544, -50.93, 107.813, -147.431, 107.786, -177.387, -1601.482]
  MoveL 883 to (58.51, 247.24, 80) mm, rotated rx -90 ry -25 rz 127.7 deg; joints [-10.156, -50.822, 107.664, -147.171, 107.866, -177.598, -1607.701]
  MoveL 884 to (58.95, 253.96, 90) mm, rotated rx -90 ry -25 rz 134.15 deg; joints [-9.769, -50.71, 107.509, -146.912, 107.945, -177.809, -1614.147]
  MoveL 885 to (58.6, 260.81, 100) mm, rotated rx -90 ry -25 rz 140.79 deg; joints [-9.383, -50.593, 107.348, -146.654, 108.024, -178.021, -1620.794]
  MoveL 886 to (57.44, 267.68, 110) mm, rotated rx -90 ry -25 rz 147.61 deg; joints [-8.998, -50.474, 107.18, -146.398, 108.101, -178.234, -1627.613]
  MoveL 887 to (55.46, 274.42, 120) mm, rotated rx -90 ry -25 rz 154.57 deg; joints [-8.614, -50.351, 107.007, -146.144, 108.175, -178.449, -1634.572]
  MoveL 888 to (52.68, 280.9, 130) mm, rotated rx -90 ry -25 rz 161.64 deg; joints [-8.231, -50.226, 106.827, -145.892, 108.247, -178.665, -1641.638]
  MoveL 889 to (49.15, 286.99, 140) mm, rotated rx -90 ry -25 rz 168.77 deg; joints [-7.849, -50.1, 106.64, -145.642, 108.316, -178.884, -1648.774]
  MoveL 890 to (44.94, 292.58, 150) mm, rotated rx -90 ry -25 rz 175.94 deg; joints [-7.468, -49.972, 106.447, -145.394, 108.381, -179.106, -1655.941]
  MoveL 891 to (40.17, 297.58, 160) mm, rotated rx -90 ry -25 rz -176.91 deg; joints [-7.088, -49.845, 106.248, -145.148, 108.442, -179.33, -1663.094]
  MoveL 892 to (34.94, 301.92, 170) mm, rotated rx -90 ry -25 rz -169.81 deg; joints [-6.709, -49.717, 106.043, -144.905, 108.498, -179.559, -1670.188]
  MoveL 893 to (29.38, 305.54, 180) mm, rotated rx -90 ry -25 rz -162.82 deg; joints [-6.332, -49.59, 105.83, -144.665, 108.55, -179.791, -1677.176]
  MoveL 894 to (23.62, 308.44, 190) mm, rotated rx -90 ry -25 rz -155.99 deg; joints [-5.956, -49.463, 105.612, -144.428, 108.597, -180.027, -1684.006]
  MoveL 895 to (17.8, 310.63, 200) mm, rotated rx -90 ry -25 rz -149.37 deg; joints [-5.581, -49.336, 105.386, -144.193, 108.639, -180.267, -1690.629]
  MoveL 896 to (12.04, 312.14, 210) mm, rotated rx -90 ry -25 rz -143.01 deg; joints [-5.207, -49.21, 105.155, -143.961, 108.676, -180.511, -1696.995]
  MoveL 897 to (6.46, 313.03, 220) mm, rotated rx -90 ry -25 rz -136.95 deg; joints [-4.834, -49.084, 104.916, -143.732, 108.709, -180.759, -1703.053]
  MoveL 898 to (1.16, 313.37, 230) mm, rotated rx -90 ry -25 rz -131.24 deg; joints [-4.463, -48.957, 104.672, -143.506, 108.737, -181.01, -1708.756]
  MoveL 899 to (-3.78, 313.26, 240) mm, rotated rx -90 ry -25 rz -125.94 deg; joints [-4.093, -48.829, 104.421, -143.282, 108.763, -181.265, -1714.059]
  MoveL 900 to (-8.28, 312.8, 250) mm, rotated rx -90 ry -25 rz -121.08 deg; joints [-3.725, -48.7, 104.163, -143.062, 108.785, -181.522, -1718.917]
  MoveL 901 to (-12.3, 312.09, 260) mm, rotated rx -90 ry -25 rz -116.71 deg; joints [-3.358, -48.569, 103.899, -142.843, 108.804, -181.783, -1723.29]
  MoveL 902 to (-15.8, 311.23, 270) mm, rotated rx -90 ry -25 rz -112.86 deg; joints [-2.992, -48.436, 103.629, -142.628, 108.822, -182.046, -1727.138]
  MoveL 903 to (-18.74, 310.33, 280) mm, rotated rx -90 ry -25 rz -109.58 deg; joints [-2.628, -48.3, 103.352, -142.414, 108.837, -182.31, -1730.424]
  MoveL 904 to (-21.11, 309.47, 290) mm, rotated rx -90 ry -25 rz -106.89 deg; joints [-2.265, -48.16, 103.069, -142.203, 108.851, -182.577, -1733.11]
  Set speed (1000.0 mm/s)
  MoveL 905 to (-21.11, 309.47, 290) mm, rotated rx -90 ry -25 rz -106.89 deg; joints [-2.265, -48.16, 103.069, -142.203, 108.851, -182.577, -1733.11]
  Set speed (1000.0 mm/s)
  MoveL 906 to (-34.79, 325.15, 290) mm, rotated rx -90 ry -25 rz -101.9 deg; joints [-2.265, -49.106, 102.979, -142.415, 108.03, -183.245, -1738.101]
  MoveL 907 to (-34.79, 325.15, 290) mm, rotated rx -90 ry -25 rz -101.9 deg; joints [-2.265, -49.106, 102.979, -142.415, 108.03, -183.245, -1738.101]
  Set speed (60.0 mm/s)
  MoveL 908 to (-31.73, 326.57, 280) mm, rotated rx -90 ry -25 rz -104.51 deg; joints [-2.628, -49.248, 103.262, -142.625, 108.013, -182.977, -1735.486]
  MoveL 909 to (-27.92, 328.13, 270) mm, rotated rx -90 ry -25 rz -107.71 deg; joints [-2.992, -49.386, 103.539, -142.837, 107.994, -182.709, -1732.288]
  MoveL 910 to (-23.38, 329.69, 260) mm, rotated rx -90 ry -25 rz -111.46 deg; joints [-3.358, -49.521, 103.809, -143.052, 107.973, -182.444, -1728.542]
  MoveL 911 to (-18.11, 331.13, 250) mm, rotated rx -90 ry -25 rz -115.71 deg; joints [-3.725, -49.652, 104.073, -143.269, 107.951, -182.18, -1724.286]
  MoveL 912 to (-12.17, 332.29, 240) mm, rotated rx -90 ry -25 rz -120.44 deg; joints [-4.093, -49.782, 104.331, -143.488, 107.926, -181.919, -1719.557]
  MoveL 913 to (-5.61, 333.04, 230) mm, rotated rx -90 ry -25 rz -125.61 deg; joints [-4.463, -49.91, 104.583, -143.711, 107.899, -181.661, -1714.392]
  MoveL 914 to (1.49, 333.22, 220) mm, rotated rx -90 ry -25 rz -131.17 deg; joints [-4.834, -50.036, 104.828, -143.935, 107.868, -181.406, -1708.834]
  MoveL 915 to (9.03, 332.72, 210) mm, rotated rx -90 ry -25 rz -137.08 deg; joints [-5.207, -50.162, 105.066, -144.163, 107.833, -181.154, -1702.922]
  MoveL 916 to (16.88, 331.41, 200) mm, rotated rx -90 ry -25 rz -143.3 deg; joints [-5.581, -50.288, 105.298, -144.393, 107.794, -180.906, -1696.702]
  MoveL 917 to (24.89, 329.2, 190) mm, rotated rx -90 ry -25 rz -149.78 deg; joints [-5.956, -50.413, 105.523, -144.626, 107.75, -180.662, -1690.217]
  MoveL 918 to (32.91, 326.04, 180) mm, rotated rx -90 ry -25 rz -156.49 deg; joints [-6.332, -50.539, 105.741, -144.861, 107.702, -180.421, -1683.513]
  MoveL 919 to (40.75, 321.89, 170) mm, rotated rx -90 ry -25 rz -163.36 deg; joints [-6.709, -50.666, 105.953, -145.1, 107.648, -180.185, -1676.637]
  MoveL 920 to (48.24, 316.75, 160) mm, rotated rx -90 ry -25 rz -170.37 deg; joints [-7.088, -50.792, 106.159, -145.341, 107.59, -179.952, -1669.635]
  MoveL 921 to (55.2, 310.67, 150) mm, rotated rx -90 ry -25 rz -177.45 deg; joints [-7.468, -50.919, 106.357, -145.584, 107.527, -179.723, -1662.551]
  MoveL 922 to (61.48, 303.74, 140) mm, rotated rx -90 ry -25 rz 175.43 deg; joints [-7.849, -51.045, 106.549, -145.83, 107.459, -179.497, -1655.431]
  MoveL 923 to (66.92, 296.06, 130) mm, rotated rx -90 ry -25 rz 168.32 deg; joints [-8.231, -51.171, 106.735, -146.078, 107.388, -179.274, -1648.317]
  MoveL 924 to (71.41, 287.77, 120) mm, rotated rx -90 ry -25 rz 161.25 deg; joints [-8.614, -51.296, 106.914, -146.329, 107.313, -179.054, -1641.249]
  MoveL 925 to (74.87, 279.04, 110) mm, rotated rx -90 ry -25 rz 154.27 deg; joints [-8.998, -51.419, 107.087, -146.581, 107.234, -178.836, -1634.266]
  MoveL 926 to (77.24, 270.04, 100) mm, rotated rx -90 ry -25 rz 147.4 deg; joints [-9.383, -51.539, 107.253, -146.835, 107.154, -178.62, -1627.404]
  MoveL 927 to (78.53, 260.95, 90) mm, rotated rx -90 ry -25 rz 140.7 deg; joints [-9.769, -51.657, 107.413, -147.091, 107.071, -178.405, -1620.696]
  MoveL 928 to (78.77, 251.96, 80) mm, rotated rx -90 ry -25 rz 134.17 deg; joints [-10.156, -51.77, 107.567, -147.348, 106.987, -178.191, -1614.174]
  MoveL 929 to (78, 243.23, 70) mm, rotated rx -90 ry -25 rz 127.87 deg; joints [-10.544, -51.88, 107.715, -147.607, 106.902, -177.977, -1607.868]
  MoveL 930 to (76.35, 234.91, 60) mm, rotated rx -90 ry -25 rz 131.81 deg; joints [-10.989, -47.633, 107.251, -146.07, 118.961, -170.899, -1601.808]
  MoveL 931 to (73.92, 227.12, 50) mm, rotated rx -90 ry -25 rz 126.02 deg; joints [-11.377, -47.728, 107.39, -146.301, 118.889, -170.685, -1596.021]
  MoveL 932 to (70.87, 219.96, 40) mm, rotated rx -90 ry -25 rz 120.54 deg; joints [-11.765, -47.818, 107.523, -146.533, 118.816, -170.472, -1590.535]
  MoveL 933 to (67.34, 213.5, 30) mm, rotated rx -90 ry -25 rz 115.38 deg; joints [-12.154, -47.902, 107.65, -146.766, 118.744, -170.258, -1585.378]
  MoveL 934 to (63.51, 207.78, 20) mm, rotated rx -90 ry -25 rz 110.58 deg; joints [-12.543, -47.981, 107.771, -147, 118.672, -170.045, -1580.576]
  MoveL 935 to (59.54, 202.81, 10) mm, rotated rx -90 ry -25 rz 106.16 deg; joints [-12.934, -48.054, 107.885, -147.235, 118.6, -169.831, -1576.157]
  MoveL 936 to (55.59, 198.58, 0) mm, rotated rx -90 ry -25 rz 102.15 deg; joints [-13.325, -48.121, 107.993, -147.471, 118.529, -169.618, -1572.15]
  Set speed (1000.0 mm/s)
  MoveL 937 to (55.59, 198.58, 0) mm, rotated rx -90 ry -25 rz 102.15 deg; joints [-13.325, -48.121, 107.993, -147.471, 118.529, -169.618, -1572.15]
  Set speed (1000.0 mm/s)
  MoveL 938 to (-34.79, 325.15, 290) mm, rotated rx -90 ry -25 rz -101.9 deg; joints [-2.265, -49.106, 102.979, -142.415, 108.03, -183.245, -1738.101]
  MoveL 939 to (-34.79, 325.15, 290) mm, rotated rx -90 ry -25 rz -101.9 deg; joints [-2.265, -49.106, 102.979, -142.415, 108.03, -183.245, -1738.101]
  Set speed (60.0 mm/s)
  MoveL 940 to (-30.72, 304.75, 290) mm, rotated rx -90 ry -25 rz -95.53 deg; joints [-2.265, -48.183, 103.068, -142.208, 108.831, -182.593, -1744.467]
  Set speed (1000.0 mm/s)
  MoveL 941 to (-30.72, 304.75, 290) mm, rotated rx -90 ry -25 rz -95.53 deg; joints [-2.265, -48.183, 103.068, -142.208, 108.831, -182.593, -1744.467]
  Set speed (1000.0 mm/s)
  MoveL 942 to (55.59, 198.58, 0) mm, rotated rx -90 ry -25 rz 102.15 deg; joints [-13.325, -48.121, 107.993, -147.471, 118.529, -169.618, -1572.15]
  MoveL 943 to (55.59, 198.58, 0) mm, rotated rx -90 ry -25 rz 102.15 deg; joints [-13.325, -48.121, 107.993, -147.471, 118.529, -169.618, -1572.15]
  Set speed (60.0 mm/s)
  MoveL 944 to (45.21, 216.6, 0) mm, rotated rx -90 ry -25 rz 96.17 deg; joints [-13.282, -51.496, 108.69, -149.277, 107.269, -175.887, -1576.169]
  Set speed (1000.0 mm/s)
  MoveL 945 to (45.21, 216.6, 0) mm, rotated rx -90 ry -25 rz 96.17 deg; joints [-13.282, -51.496, 108.69, -149.277, 107.269, -175.887, -1576.169]
  Set speed (1000.0 mm/s)
  MoveL 946 to (55.59, 198.58, 0) mm, rotated rx -90 ry -25 rz 102.15 deg; joints [-13.325, -48.121, 107.993, -147.471, 118.529, -169.618, -1572.15]
  MoveL 947 to (55.59, 198.58, 0) mm, rotated rx -90 ry -25 rz 102.15 deg; joints [-13.325, -48.121, 107.993, -147.471, 118.529, -169.618, -1572.15]
  Set speed (60.0 mm/s)
  MoveL 948 to (59.54, 202.81, 10) mm, rotated rx -90 ry -25 rz 106.16 deg; joints [-12.934, -48.054, 107.885, -147.235, 118.6, -169.831, -1576.157]
  MoveL 949 to (63.51, 207.78, 20) mm, rotated rx -90 ry -25 rz 110.58 deg; joints [-12.543, -47.981, 107.771, -147, 118.672, -170.045, -1580.576]
  MoveL 950 to (67.34, 213.5, 30) mm, rotated rx -90 ry -25 rz 115.38 deg; joints [-12.154, -47.902, 107.65, -146.766, 118.744, -170.258, -1585.378]
  MoveL 951 to (70.87, 219.96, 40) mm, rotated rx -90 ry -25 rz 120.54 deg; joints [-11.765, -47.818, 107.523, -146.533, 118.816, -170.472, -1590.535]
  MoveL 952 to (73.92, 227.12, 50) mm, rotated rx -90 ry -25 rz 126.02 deg; joints [-11.377, -47.728, 107.39, -146.301, 118.889, -170.685, -1596.021]
  MoveL 953 to (76.35, 234.91, 60) mm, rotated rx -90 ry -25 rz 131.81 deg; joints [-10.989, -47.633, 107.251, -146.07, 118.961, -170.899, -1601.808]
  MoveL 954 to (78, 243.23, 70) mm, rotated rx -90 ry -25 rz 127.87 deg; joints [-10.544, -51.88, 107.715, -147.607, 106.902, -177.977, -1607.868]
  MoveL 955 to (78.77, 251.96, 80) mm, rotated rx -90 ry -25 rz 134.17 deg; joints [-10.156, -51.77, 107.567, -147.348, 106.987, -178.191, -1614.174]
  MoveL 956 to (78.53, 260.95, 90) mm, rotated rx -90 ry -25 rz 140.7 deg; joints [-9.769, -51.657, 107.413, -147.091, 107.071, -178.405, -1620.696]
  MoveL 957 to (77.24, 270.04, 100) mm, rotated rx -90 ry -25 rz 147.4 deg; joints [-9.383, -51.539, 107.253, -146.835, 107.154, -178.62, -1627.404]
  MoveL 958 to (74.87, 279.04, 110) mm, rotated rx -90 ry -25 rz 154.27 deg; joints [-8.998, -51.419, 107.087, -146.581, 107.234, -178.836, -1634.266]
  MoveL 959 to (71.41, 287.77, 120) mm, rotated rx -90 ry -25 rz 161.25 deg; joints [-8.614, -51.296, 106.914, -146.329, 107.313, -179.054, -1641.249]
  MoveL 960 to (66.92, 296.06, 130) mm, rotated rx -90 ry -25 rz 168.32 deg; joints [-8.231, -51.171, 106.735, -146.078, 107.388, -179.274, -1648.317]
  MoveL 961 to (61.48, 303.74, 140) mm, rotated rx -90 ry -25 rz 175.43 deg; joints [-7.849, -51.045, 106.549, -145.83, 107.459, -179.497, -1655.431]
  MoveL 962 to (55.2, 310.67, 150) mm, rotated rx -90 ry -25 rz -177.45 deg; joints [-7.468, -50.919, 106.357, -145.584, 107.527, -179.723, -1662.551]
  MoveL 963 to (48.24, 316.75, 160) mm, rotated rx -90 ry -25 rz -170.37 deg; joints [-7.088, -50.792, 106.159, -145.341, 107.59, -179.952, -1669.635]
  MoveL 964 to (40.75, 321.89, 170) mm, rotated rx -90 ry -25 rz -163.36 deg; joints [-6.709, -50.666, 105.953, -145.1, 107.648, -180.185, -1676.637]
  MoveL 965 to (32.91, 326.04, 180) mm, rotated rx -90 ry -25 rz -156.49 deg; joints [-6.332, -50.539, 105.741, -144.861, 107.702, -180.421, -1683.513]
  MoveL 966 to (24.89, 329.2, 190) mm, rotated rx -90 ry -25 rz -149.78 deg; joints [-5.956, -50.413, 105.523, -144.626, 107.75, -180.662, -1690.217]
  MoveL 967 to (16.88, 331.41, 200) mm, rotated rx -90 ry -25 rz -143.3 deg; joints [-5.581, -50.288, 105.298, -144.393, 107.794, -180.906, -1696.702]
  MoveL 968 to (9.03, 332.72, 210) mm, rotated rx -90 ry -25 rz -137.08 deg; joints [-5.207, -50.162, 105.066, -144.163, 107.833, -181.154, -1702.922]
  MoveL 969 to (1.49, 333.22, 220) mm, rotated rx -90 ry -25 rz -131.17 deg; joints [-4.834, -50.036, 104.828, -143.935, 107.868, -181.406, -1708.834]
  MoveL 970 to (-5.61, 333.04, 230) mm, rotated rx -90 ry -25 rz -125.61 deg; joints [-4.463, -49.91, 104.583, -143.711, 107.899, -181.661, -1714.392]
  MoveL 971 to (-12.17, 332.29, 240) mm, rotated rx -90 ry -25 rz -120.44 deg; joints [-4.093, -49.782, 104.331, -143.488, 107.926, -181.919, -1719.557]
  MoveL 972 to (-18.11, 331.13, 250) mm, rotated rx -90 ry -25 rz -115.71 deg; joints [-3.725, -49.652, 104.073, -143.269, 107.951, -182.18, -1724.286]
  MoveL 973 to (-23.38, 329.69, 260) mm, rotated rx -90 ry -25 rz -111.46 deg; joints [-3.358, -49.521, 103.809, -143.052, 107.973, -182.444, -1728.542]
  MoveL 974 to (-27.92, 328.13, 270) mm, rotated rx -90 ry -25 rz -107.71 deg; joints [-2.992, -49.386, 103.539, -142.837, 107.994, -182.709, -1732.288]
  MoveL 975 to (-31.73, 326.57, 280) mm, rotated rx -90 ry -25 rz -104.51 deg; joints [-2.628, -49.248, 103.262, -142.625, 108.013, -182.977, -1735.486]
  MoveL 976 to (-34.79, 325.15, 290) mm, rotated rx -90 ry -25 rz -101.9 deg; joints [-2.265, -49.106, 102.979, -142.415, 108.03, -183.245, -1738.101]
  Set speed (1000.0 mm/s)
  MoveL 977 to (-34.79, 325.15, 290) mm, rotated rx -90 ry -25 rz -101.9 deg; joints [-2.265, -49.106, 102.979, -142.415, 108.03, -183.245, -1738.101]
  Set speed (1000.0 mm/s)
  MoveL 978 to (-30.72, 304.75, 290) mm, rotated rx -90 ry -25 rz -95.53 deg; joints [-2.265, -48.183, 103.068, -142.208, 108.831, -182.593, -1744.467]
  MoveL 979 to (-30.72, 304.75, 290) mm, rotated rx -90 ry -25 rz -95.53 deg; joints [-2.265, -48.183, 103.068, -142.208, 108.831, -182.593, -1744.467]
  Set speed (60.0 mm/s)
  MoveL 980 to (-28.54, 306.02, 280) mm, rotated rx -90 ry -25 rz -98.19 deg; joints [-2.628, -48.321, 103.351, -142.419, 108.819, -182.325, -1741.806]
  MoveL 981 to (-25.81, 307.44, 270) mm, rotated rx -90 ry -25 rz -101.45 deg; joints [-2.992, -48.455, 103.627, -142.632, 108.805, -182.059, -1738.548]
  MoveL 982 to (-22.53, 308.91, 260) mm, rotated rx -90 ry -25 rz -105.27 deg; joints [-3.358, -48.585, 103.898, -142.847, 108.791, -181.794, -1734.728]
  MoveL 983 to (-18.7, 310.34, 250) mm, rotated rx -90 ry -25 rz -109.62 deg; joints [-3.725, -48.713, 104.162, -143.064, 108.774, -181.531, -1730.381]
  MoveL 984 to (-14.35, 311.61, 240) mm, rotated rx -90 ry -25 rz -114.46 deg; joints [-4.093, -48.838, 104.42, -143.284, 108.756, -181.27, -1725.543]
  MoveL 985 to (-9.52, 312.61, 230) mm, rotated rx -90 ry -25 rz -119.75 deg; joints [-4.463, -48.961, 104.671, -143.507, 108.734, -181.013, -1720.254]
  MoveL 986 to (-4.24, 313.23, 220) mm, rotated rx -90 ry -25 rz -125.45 deg; joints [-4.834, -49.083, 104.916, -143.732, 108.71, -180.758, -1714.554]
  MoveL 987 to (1.41, 313.37, 210) mm, rotated rx -90 ry -25 rz -131.51 deg; joints [-5.207, -49.204, 105.155, -143.96, 108.681, -180.507, -1708.487]
  MoveL 988 to (7.35, 312.92, 200) mm, rotated rx -90 ry -25 rz -137.9 deg; joints [-5.581, -49.324, 105.387, -144.19, 108.649, -180.259, -1702.098]
  MoveL 989 to (13.47, 311.83, 190) mm, rotated rx -90 ry -25 rz -144.57 deg; joints [-5.956, -49.446, 105.613, -144.424, 108.612, -180.016, -1695.435]
  MoveL 990 to (19.65, 310.01, 180) mm, rotated rx -90 ry -25 rz -151.45 deg; joints [-6.332, -49.567, 105.832, -144.66, 108.57, -179.776, -1688.548]
  MoveL 991 to (25.78, 307.45, 170) mm, rotated rx -90 ry -25 rz -158.51 deg; joints [-6.709, -49.689, 106.045, -144.9, 108.523, -179.54, -1681.489]
  MoveL 992 to (31.7, 304.13, 160) mm, rotated rx -90 ry -25 rz -165.69 deg; joints [-7.088, -49.812, 106.251, -145.141, 108.471, -179.309, -1674.307]
  MoveL 993 to (37.3, 300.08, 150) mm, rotated rx -90 ry -25 rz -172.95 deg; joints [-7.468, -49.935, 106.45, -145.386, 108.414, -179.081, -1667.054]
  MoveL 994 to (42.45, 295.34, 140) mm, rotated rx -90 ry -25 rz 179.78 deg; joints [-7.849, -50.059, 106.643, -145.633, 108.353, -178.858, -1659.778]
  MoveL 995 to (47.02, 289.99, 130) mm, rotated rx -90 ry -25 rz 172.52 deg; joints [-8.231, -50.182, 106.83, -145.883, 108.287, -178.637, -1652.524]
  MoveL 996 to (50.93, 284.12, 120) mm, rotated rx -90 ry -25 rz 165.34 deg; joints [-8.614, -50.304, 107.01, -146.135, 108.218, -178.419, -1645.337]
  MoveL 997 to (54.1, 277.85, 110) mm, rotated rx -90 ry -25 rz 158.26 deg; joints [-8.998, -50.425, 107.184, -146.389, 108.145, -178.204, -1638.256]
  MoveL 998 to (56.49, 271.3, 100) mm, rotated rx -90 ry -25 rz 151.32 deg; joints [-9.383, -50.544, 107.352, -146.645, 108.069, -177.99, -1631.316]
  MoveL 999 to (58.06, 264.62, 90) mm, rotated rx -90 ry -25 rz 144.55 deg; joints [-9.769, -50.66, 107.513, -146.902, 107.991, -177.778, -1624.553]
  MoveL 1000 to (58.85, 257.94, 80) mm, rotated rx -90 ry -25 rz 138 deg; joints [-10.156, -50.772, 107.668, -147.161, 107.911, -177.567, -1617.997]
  MoveL 1001 to (58.87, 251.39, 70) mm, rotated rx -90 ry -25 rz 131.68 deg; joints [-10.544, -50.881, 107.817, -147.422, 107.831, -177.357, -1611.675]
  MoveL 1002 to (58.2, 245.07, 60) mm, rotated rx -90 ry -25 rz 125.62 deg; joints [-10.933, -50.985, 107.96, -147.684, 107.75, -177.148, -1605.616]
  MoveL 1003 to (56.92, 239.11, 50) mm, rotated rx -90 ry -25 rz 119.84 deg; joints [-11.323, -51.084, 108.096, -147.947, 107.669, -176.938, -1599.845]
  MoveL 1004 to (55.13, 233.57, 40) mm, rotated rx -90 ry -25 rz 114.39 deg; joints [-11.713, -51.178, 108.227, -148.211, 107.588, -176.728, -1594.385]
  MoveL 1005 to (52.95, 228.52, 30) mm, rotated rx -90 ry -25 rz 109.26 deg; joints [-12.104, -51.266, 108.352, -148.476, 107.507, -176.518, -1589.263]
  MoveL 1006 to (50.48, 223.99, 20) mm, rotated rx -90 ry -25 rz 104.5 deg; joints [-12.496, -51.348, 108.47, -148.742, 107.427, -176.308, -1584.503]
  MoveL 1007 to (47.86, 220.02, 10) mm, rotated rx -90 ry -25 rz 100.13 deg; joints [-12.889, -51.425, 108.583, -149.009, 107.348, -176.097, -1580.13]
  MoveL 1008 to (45.21, 216.6, 0) mm, rotated rx -90 ry -25 rz 96.17 deg; joints [-13.282, -51.496, 108.69, -149.277, 107.269, -175.887, -1576.169]
  Set speed (1000.0 mm/s)
  MoveL 1009 to (45.21, 216.6, 0) mm, rotated rx -90 ry -25 rz 96.17 deg; joints [-13.282, -51.496, 108.69, -149.277, 107.269, -175.887, -1576.169]
  Set speed (1000.0 mm/s)
  MoveL 1010 to (-30.72, 304.75, 290) mm, rotated rx -90 ry -25 rz -95.53 deg; joints [-2.265, -48.183, 103.068, -142.208, 108.831, -182.593, -1744.467]
  MoveL 1011 to (-30.72, 304.75, 290) mm, rotated rx -90 ry -25 rz -95.53 deg; joints [-2.265, -48.183, 103.068, -142.208, 108.831, -182.593, -1744.467]
  Set speed (60.0 mm/s)
  MoveL 1012 to (-58.22, 263.67, 290) mm, rotated rx -90 ry -25 rz -43.61 deg; joints [-2.265, -48.376, 103.052, -142.252, 108.666, -182.728, -1796.394]
  Set speed (1000.0 mm/s)
  MoveL 1013 to (-58.22, 263.67, 290) mm, rotated rx -90 ry -25 rz -43.61 deg; joints [-2.265, -48.376, 103.052, -142.252, 108.666, -182.728, -1796.394]
  Set speed (1000.0 mm/s)
  MoveL 1014 to (45.21, 216.6, 0) mm, rotated rx -90 ry -25 rz 96.17 deg; joints [-13.282, -51.496, 108.69, -149.277, 107.269, -175.887, -1936.169]
  MoveL 1015 to (45.21, 216.6, 0) mm, rotated rx -90 ry -25 rz 96.17 deg; joints [-13.282, -51.496, 108.69, -149.277, 107.269, -175.887, -1936.169]
  Set speed (60.0 mm/s)
  MoveL 1016 to (58.12, 264.32, 0) mm, rotated rx -90 ry -25 rz 144.25 deg; joints [-13.282, -51.276, 108.708, -149.239, 107.474, -175.759, -1984.254]
  Set speed (1000.0 mm/s)
  MoveL 1017 to (58.12, 264.32, 0) mm, rotated rx -90 ry -25 rz 144.25 deg; joints [-13.282, -51.276, 108.708, -149.239, 107.474, -175.759, -1984.254]
  Set speed (1000.0 mm/s)
  MoveL 1018 to (45.21, 216.6, 0) mm, rotated rx -90 ry -25 rz 96.17 deg; joints [-13.282, -51.496, 108.69, -149.277, 107.269, -175.887, -1936.169]
  MoveL 1019 to (45.21, 216.6, 0) mm, rotated rx -90 ry -25 rz 96.17 deg; joints [-13.282, -51.496, 108.69, -149.277, 107.269, -175.887, -1936.169]
  Set speed (60.0 mm/s)
  MoveL 1020 to (47.86, 220.02, 10) mm, rotated rx -90 ry -25 rz 100.13 deg; joints [-12.889, -51.425, 108.583, -149.009, 107.348, -176.097, -1940.13]
  MoveL 1021 to (50.48, 223.99, 20) mm, rotated rx -90 ry -25 rz 104.5 deg; joints [-12.496, -51.348, 108.47, -148.742, 107.427, -176.308, -1944.503]
  MoveL 1022 to (52.95, 228.52, 30) mm, rotated rx -90 ry -25 rz 109.26 deg; joints [-12.104, -51.266, 108.352, -148.476, 107.507, -176.518, -1949.263]
  MoveL 1023 to (55.13, 233.57, 40) mm, rotated rx -90 ry -25 rz 114.39 deg; joints [-11.713, -51.178, 108.227, -148.211, 107.588, -176.728, -1954.385]
  MoveL 1024 to (56.92, 239.11, 50) mm, rotated rx -90 ry -25 rz 119.84 deg; joints [-11.323, -51.084, 108.096, -147.947, 107.669, -176.938, -1959.845]
  MoveL 1025 to (58.2, 245.07, 60) mm, rotated rx -90 ry -25 rz 125.62 deg; joints [-10.933, -50.985, 107.96, -147.684, 107.75, -177.148, -1965.616]
  MoveL 1026 to (58.87, 251.39, 70) mm, rotated rx -90 ry -25 rz 131.68 deg; joints [-10.544, -50.881, 107.817, -147.422, 107.831, -177.357, -1971.675]
  MoveL 1027 to (58.85, 257.94, 80) mm, rotated rx -90 ry -25 rz 138 deg; joints [-10.156, -50.772, 107.668, -147.161, 107.911, -177.567, -1977.997]
  MoveL 1028 to (58.06, 264.62, 90) mm, rotated rx -90 ry -25 rz 144.55 deg; joints [-9.769, -50.66, 107.513, -146.902, 107.991, -177.778, -1984.553]
  MoveL 1029 to (56.49, 271.3, 100) mm, rotated rx -90 ry -25 rz 151.32 deg; joints [-9.383, -50.544, 107.352, -146.645, 108.069, -177.99, -1991.316]
  MoveL 1030 to (54.1, 277.85, 110) mm, rotated rx -90 ry -25 rz 158.26 deg; joints [-8.998, -50.425, 107.184, -146.389, 108.145, -178.204, -1998.256]
  MoveL 1031 to (50.93, 284.12, 120) mm, rotated rx -90 ry -25 rz 165.34 deg; joints [-8.614, -50.304, 107.01, -146.135, 108.218, -178.419, -2005.337]
  MoveL 1032 to (47.02, 289.99, 130) mm, rotated rx -90 ry -25 rz 172.52 deg; joints [-8.231, -50.182, 106.83, -145.883, 108.287, -178.637, -2012.524]
  MoveL 1033 to (42.45, 295.34, 140) mm, rotated rx -90 ry -25 rz 179.78 deg; joints [-7.849, -50.059, 106.643, -145.633, 108.353, -178.858, -2019.778]
  MoveL 1034 to (37.3, 300.08, 150) mm, rotated rx -90 ry -25 rz -172.95 deg; joints [-7.468, -49.935, 106.45, -145.386, 108.414, -179.081, -2027.054]
  MoveL 1035 to (31.7, 304.13, 160) mm, rotated rx -90 ry -25 rz -165.69 deg; joints [-7.088, -49.812, 106.251, -145.141, 108.471, -179.309, -2034.307]
  MoveL 1036 to (25.78, 307.45, 170) mm, rotated rx -90 ry -25 rz -158.51 deg; joints [-6.709, -49.689, 106.045, -144.9, 108.523, -179.54, -2041.489]
  MoveL 1037 to (19.65, 310.01, 180) mm, rotated rx -90 ry -25 rz -151.45 deg; joints [-6.332, -49.567, 105.832, -144.66, 108.57, -179.776, -2048.548]
  MoveL 1038 to (13.47, 311.83, 190) mm, rotated rx -90 ry -25 rz -144.57 deg; joints [-5.956, -49.446, 105.613, -144.424, 108.612, -180.016, -2055.435]
  MoveL 1039 to (7.35, 312.92, 200) mm, rotated rx -90 ry -25 rz -137.9 deg; joints [-5.581, -49.324, 105.387, -144.19, 108.649, -180.259, -2062.098]
  MoveL 1040 to (1.41, 313.37, 210) mm, rotated rx -90 ry -25 rz -131.51 deg; joints [-5.207, -49.204, 105.155, -143.96, 108.681, -180.507, -2068.487]
  MoveL 1041 to (-4.24, 313.23, 220) mm, rotated rx -90 ry -25 rz -125.45 deg; joints [-4.834, -49.083, 104.916, -143.732, 108.71, -180.758, -2074.554]
  MoveL 1042 to (-9.52, 312.61, 230) mm, rotated rx -90 ry -25 rz -119.75 deg; joints [-4.463, -48.961, 104.671, -143.507, 108.734, -181.013, -2080.254]
  MoveL 1043 to (-14.35, 311.61, 240) mm, rotated rx -90 ry -25 rz -114.46 deg; joints [-4.093, -48.838, 104.42, -143.284, 108.756, -181.27, -2085.543]
  MoveL 1044 to (-18.7, 310.34, 250) mm, rotated rx -90 ry -25 rz -109.62 deg; joints [-3.725, -48.713, 104.162, -143.064, 108.774, -181.531, -2090.381]
  MoveL 1045 to (-22.53, 308.91, 260) mm, rotated rx -90 ry -25 rz -105.27 deg; joints [-3.358, -48.585, 103.898, -142.847, 108.791, -181.794, -2094.728]
  MoveL 1046 to (-25.81, 307.44, 270) mm, rotated rx -90 ry -25 rz -101.45 deg; joints [-2.992, -48.455, 103.627, -142.632, 108.805, -182.059, -2098.548]
  MoveL 1047 to (-28.54, 306.02, 280) mm, rotated rx -90 ry -25 rz -98.19 deg; joints [-2.628, -48.321, 103.351, -142.419, 108.819, -182.325, -2101.806]
  MoveL 1048 to (-30.72, 304.75, 290) mm, rotated rx -90 ry -25 rz -95.53 deg; joints [-2.265, -48.183, 103.068, -142.208, 108.831, -182.593, -2104.467]
  Set speed (1000.0 mm/s)
  MoveL 1049 to (-30.72, 304.75, 290) mm, rotated rx -90 ry -25 rz -95.53 deg; joints [-2.265, -48.183, 103.068, -142.208, 108.831, -182.593, -2104.467]
  Set speed (1000.0 mm/s)
  MoveL 1050 to (-58.22, 263.67, 290) mm, rotated rx -90 ry -25 rz -43.61 deg; joints [-2.265, -48.376, 103.052, -142.252, 108.666, -182.728, -2156.394]
  MoveL 1051 to (-58.22, 263.67, 290) mm, rotated rx -90 ry -25 rz -43.61 deg; joints [-2.265, -48.376, 103.052, -142.252, 108.666, -182.728, -2156.394]
  Set speed (60.0 mm/s)
  MoveL 1052 to (-57.77, 266.15, 280) mm, rotated rx -90 ry -25 rz -46.08 deg; joints [-2.628, -48.509, 103.335, -142.461, 108.657, -182.456, -2153.924]
  MoveL 1053 to (-57.08, 269.15, 270) mm, rotated rx -90 ry -25 rz -49.11 deg; joints [-2.992, -48.637, 103.613, -142.672, 108.649, -182.185, -2150.894]
  MoveL 1054 to (-56.08, 272.6, 260) mm, rotated rx -90 ry -25 rz -52.67 deg; joints [-3.358, -48.759, 103.884, -142.885, 108.641, -181.914, -2147.333]
  MoveL 1055 to (-54.69, 276.44, 250) mm, rotated rx -90 ry -25 rz -56.73 deg; joints [-3.725, -48.876, 104.149, -143.1, 108.633, -181.643, -2143.267]
  MoveL 1056 to (-52.84, 280.57, 240) mm, rotated rx -90 ry -25 rz -61.28 deg; joints [-4.093, -48.989, 104.408, -143.317, 108.625, -181.373, -2138.724]
  MoveL 1057 to (-50.46, 284.91, 230) mm, rotated rx -90 ry -25 rz -66.27 deg; joints [-4.463, -49.097, 104.661, -143.536, 108.616, -181.105, -2133.731]
  MoveL 1058 to (-47.51, 289.33, 220) mm, rotated rx -90 ry -25 rz -71.68 deg; joints [-4.834, -49.201, 104.907, -143.757, 108.607, -180.837, -2128.316]
  MoveL 1059 to (-43.95, 293.72, 210) mm, rotated rx -90 ry -25 rz -77.49 deg; joints [-5.207, -49.301, 105.148, -143.981, 108.596, -180.572, -2122.509]
  MoveL 1060 to (-39.77, 297.95, 200) mm, rotated rx -90 ry -25 rz -83.66 deg; joints [-5.581, -49.399, 105.381, -144.206, 108.583, -180.309, -2116.342]
  MoveL 1061 to (-34.96, 301.9, 190) mm, rotated rx -90 ry -25 rz -90.15 deg; joints [-5.956, -49.495, 105.609, -144.434, 108.568, -180.048, -2109.847]
  MoveL 1062 to (-29.57, 305.43, 180) mm, rotated rx -90 ry -25 rz -96.94 deg; joints [-6.332, -49.59, 105.83, -144.665, 108.55, -179.791, -2103.063]
  MoveL 1063 to (-23.65, 308.43, 170) mm, rotated rx -90 ry -25 rz -103.97 deg; joints [-6.709, -49.684, 106.045, -144.898, 108.527, -179.537, -2096.03]
  MoveL 1064 to (-17.28, 310.79, 160) mm, rotated rx -90 ry -25 rz -111.21 deg; joints [-7.088, -49.778, 106.253, -145.135, 108.501, -179.287, -2088.791]
  MoveL 1065 to (-10.57, 312.43, 150) mm, rotated rx -90 ry -25 rz -118.61 deg; joints [-7.468, -49.873, 106.455, -145.373, 108.47, -179.041, -2081.395]
  MoveL 1066 to (-3.62, 313.27, 140) mm, rotated rx -90 ry -25 rz -126.11 deg; joints [-7.849, -49.968, 106.65, -145.615, 108.433, -178.799, -2073.889]
  MoveL 1067 to (3.42, 313.28, 130) mm, rotated rx -90 ry -25 rz -133.67 deg; joints [-8.231, -50.064, 106.839, -145.859, 108.392, -178.562, -2066.327]
  MoveL 1068 to (10.42, 312.45, 120) mm, rotated rx -90 ry -25 rz -141.24 deg; joints [-8.614, -50.162, 107.021, -146.107, 108.345, -178.329, -2058.761]
  MoveL 1069 to (17.25, 310.8, 110) mm, rotated rx -90 ry -25 rz -148.76 deg; joints [-8.998, -50.261, 107.197, -146.356, 108.292, -178.1, -2051.243]
  MoveL 1070 to (23.78, 308.38, 100) mm, rotated rx -90 ry -25 rz -156.18 deg; joints [-9.383, -50.36, 107.366, -146.609, 108.234, -177.876, -2043.825]
  MoveL 1071 to (29.89, 305.25, 90) mm, rotated rx -90 ry -25 rz -163.45 deg; joints [-9.769, -50.46, 107.529, -146.864, 108.171, -177.654, -2036.554]
  MoveL 1072 to (35.48, 301.51, 80) mm, rotated rx -90 ry -25 rz -170.52 deg; joints [-10.156, -50.56, 107.685, -147.121, 108.104, -177.437, -2029.477]
  MoveL 1073 to (40.49, 297.28, 70) mm, rotated rx -90 ry -25 rz -177.36 deg; joints [-10.544, -50.659, 107.835, -147.38, 108.033, -177.221, -2022.636]
  MoveL 1074 to (44.86, 292.68, 60) mm, rotated rx -90 ry -25 rz 176.07 deg; joints [-10.933, -50.756, 107.978, -147.641, 107.959, -177.009, -2016.069]
  MoveL 1075 to (48.58, 287.83, 50) mm, rotated rx -90 ry -25 rz 169.81 deg; joints [-11.323, -50.852, 108.115, -147.904, 107.882, -176.798, -2009.813]
  MoveL 1076 to (51.63, 282.88, 40) mm, rotated rx -90 ry -25 rz 163.9 deg; joints [-11.713, -50.944, 108.246, -148.168, 107.802, -176.589, -2003.9]
  MoveL 1077 to (54.06, 277.94, 30) mm, rotated rx -90 ry -25 rz 158.36 deg; joints [-12.104, -51.034, 108.371, -148.434, 107.721, -176.38, -1998.36]
  MoveL 1078 to (55.91, 273.13, 20) mm, rotated rx -90 ry -25 rz 153.22 deg; joints [-12.496, -51.119, 108.49, -148.701, 107.639, -176.173, -1993.221]
  MoveL 1079 to (57.23, 268.56, 10) mm, rotated rx -90 ry -25 rz 148.51 deg; joints [-12.889, -51.2, 108.602, -148.969, 107.557, -175.966, -1988.51]
  MoveL 1080 to (58.12, 264.32, 0) mm, rotated rx -90 ry -25 rz 144.25 deg; joints [-13.282, -51.276, 108.708, -149.239, 107.474, -175.759, -1984.254]
  Set speed (1000.0 mm/s)
  MoveL 1081 to (58.12, 264.32, 0) mm, rotated rx -90 ry -25 rz 144.25 deg; joints [-13.282, -51.276, 108.708, -149.239, 107.474, -175.759, -1984.254]
  Set speed (1000.0 mm/s)
  MoveL 1082 to (-58.22, 263.67, 290) mm, rotated rx -90 ry -25 rz -43.61 deg; joints [-2.265, -48.376, 103.052, -142.252, 108.666, -182.728, -2156.394]
  MoveL 1083 to (-58.22, 263.67, 290) mm, rotated rx -90 ry -25 rz -43.61 deg; joints [-2.265, -48.376, 103.052, -142.252, 108.666, -182.728, -2156.394]
  Set speed (60.0 mm/s)
  MoveL 1084 to (-78.63, 259.66, 290) mm, rotated rx -90 ry -25 rz -39.75 deg; joints [-2.265, -49.329, 102.952, -142.464, 107.833, -183.405, -2160.245]
  Set speed (1000.0 mm/s)
  MoveL 1085 to (-78.63, 259.66, 290) mm, rotated rx -90 ry -25 rz -39.75 deg; joints [-2.265, -49.329, 102.952, -142.464, 107.833, -183.405, -2160.245]
  Set speed (1000.0 mm/s)
  MoveL 1086 to (58.12, 264.32, 0) mm, rotated rx -90 ry -25 rz 144.25 deg; joints [-13.282, -51.276, 108.708, -149.239, 107.474, -175.759, -1984.254]
  MoveL 1087 to (58.12, 264.32, 0) mm, rotated rx -90 ry -25 rz 144.25 deg; joints [-13.282, -51.276, 108.708, -149.239, 107.474, -175.759, -1984.254]
  Set speed (60.0 mm/s)
  MoveL 1088 to (76.17, 274.65, 0) mm, rotated rx -90 ry -25 rz 160.89 deg; joints [-13.325, -47.846, 107.991, -147.391, 118.758, -169.451, -1990.889]
  Set speed (1000.0 mm/s)
  MoveL 1089 to (76.17, 274.65, 0) mm, rotated rx -90 ry -25 rz 160.89 deg; joints [-13.325, -47.846, 107.991, -147.391, 118.758, -169.451, -1990.889]
  Set speed (1000.0 mm/s)
  MoveL 1090 to (58.12, 264.32, 0) mm, rotated rx -90 ry -25 rz 144.25 deg; joints [-13.282, -51.276, 108.708, -149.239, 107.474, -175.759, -1984.254]
  MoveL 1091 to (58.12, 264.32, 0) mm, rotated rx -90 ry -25 rz 144.25 deg; joints [-13.282, -51.276, 108.708, -149.239, 107.474, -175.759, -1984.254]
  Set speed (60.0 mm/s)
  MoveL 1092 to (57.23, 268.56, 10) mm, rotated rx -90 ry -25 rz 148.51 deg; joints [-12.889, -51.2, 108.602, -148.969, 107.557, -175.966, -1988.51]
  MoveL 1093 to (55.91, 273.13, 20) mm, rotated rx -90 ry -25 rz 153.22 deg; joints [-12.496, -51.119, 108.49, -148.701, 107.639, -176.173, -1993.221]
  MoveL 1094 to (54.06, 277.94, 30) mm, rotated rx -90 ry -25 rz 158.36 deg; joints [-12.104, -51.034, 108.371, -148.434, 107.721, -176.38, -1998.36]
  MoveL 1095 to (51.63, 282.88, 40) mm, rotated rx -90 ry -25 rz 163.9 deg; joints [-11.713, -50.944, 108.246, -148.168, 107.802, -176.589, -2003.9]
  MoveL 1096 to (48.58, 287.83, 50) mm, rotated rx -90 ry -25 rz 169.81 deg; joints [-11.323, -50.852, 108.115, -147.904, 107.882, -176.798, -2009.813]
  MoveL 1097 to (44.86, 292.68, 60) mm, rotated rx -90 ry -25 rz 176.07 deg; joints [-10.933, -50.756, 107.978, -147.641, 107.959, -177.009, -2016.069]
  MoveL 1098 to (40.49, 297.28, 70) mm, rotated rx -90 ry -25 rz -177.36 deg; joints [-10.544, -50.659, 107.835, -147.38, 108.033, -177.221, -2022.636]
  MoveL 1099 to (35.48, 301.51, 80) mm, rotated rx -90 ry -25 rz -170.52 deg; joints [-10.156, -50.56, 107.685, -147.121, 108.104, -177.437, -2029.477]
  MoveL 1100 to (29.89, 305.25, 90) mm, rotated rx -90 ry -25 rz -163.45 deg; joints [-9.769, -50.46, 107.529, -146.864, 108.171, -177.654, -2036.554]
  MoveL 1101 to (23.78, 308.38, 100) mm, rotated rx -90 ry -25 rz -156.18 deg; joints [-9.383, -50.36, 107.366, -146.609, 108.234, -177.876, -2043.825]
  MoveL 1102 to (17.25, 310.8, 110) mm, rotated rx -90 ry -25 rz -148.76 deg; joints [-8.998, -50.261, 107.197, -146.356, 108.292, -178.1, -2051.243]
  MoveL 1103 to (10.42, 312.45, 120) mm, rotated rx -90 ry -25 rz -141.24 deg; joints [-8.614, -50.162, 107.021, -146.107, 108.345, -178.329, -2058.761]
  MoveL 1104 to (3.42, 313.28, 130) mm, rotated rx -90 ry -25 rz -133.67 deg; joints [-8.231, -50.064, 106.839, -145.859, 108.392, -178.562, -2066.327]
  MoveL 1105 to (-3.62, 313.27, 140) mm, rotated rx -90 ry -25 rz -126.11 deg; joints [-7.849, -49.968, 106.65, -145.615, 108.433, -178.799, -2073.889]
  MoveL 1106 to (-10.57, 312.43, 150) mm, rotated rx -90 ry -25 rz -118.61 deg; joints [-7.468, -49.873, 106.455, -145.373, 108.47, -179.041, -2081.395]
  MoveL 1107 to (-17.28, 310.79, 160) mm, rotated rx -90 ry -25 rz -111.21 deg; joints [-7.088, -49.778, 106.253, -145.135, 108.501, -179.287, -2088.791]
  MoveL 1108 to (-23.65, 308.43, 170) mm, rotated rx -90 ry -25 rz -103.97 deg; joints [-6.709, -49.684, 106.045, -144.898, 108.527, -179.537, -2096.03]
  MoveL 1109 to (-29.57, 305.43, 180) mm, rotated rx -90 ry -25 rz -96.94 deg; joints [-6.332, -49.59, 105.83, -144.665, 108.55, -179.791, -2103.063]
  MoveL 1110 to (-34.96, 301.9, 190) mm, rotated rx -90 ry -25 rz -90.15 deg; joints [-5.956, -49.495, 105.609, -144.434, 108.568, -180.048, -2109.847]
  MoveL 1111 to (-39.77, 297.95, 200) mm, rotated rx -90 ry -25 rz -83.66 deg; joints [-5.581, -49.399, 105.381, -144.206, 108.583, -180.309, -2116.342]
  MoveL 1112 to (-43.95, 293.72, 210) mm, rotated rx -90 ry -25 rz -77.49 deg; joints [-5.207, -49.301, 105.148, -143.981, 108.596, -180.572, -2122.509]
  MoveL 1113 to (-47.51, 289.33, 220) mm, rotated rx -90 ry -25 rz -71.68 deg; joints [-4.834, -49.201, 104.907, -143.757, 108.607, -180.837, -2128.316]
  MoveL 1114 to (-50.46, 284.91, 230) mm, rotated rx -90 ry -25 rz -66.27 deg; joints [-4.463, -49.097, 104.661, -143.536, 108.616, -181.105, -2133.731]
  MoveL 1115 to (-52.84, 280.57, 240) mm, rotated rx -90 ry -25 rz -61.28 deg; joints [-4.093, -48.989, 104.408, -143.317, 108.625, -181.373, -2138.724]
  MoveL 1116 to (-54.69, 276.44, 250) mm, rotated rx -90 ry -25 rz -56.73 deg; joints [-3.725, -48.876, 104.149, -143.1, 108.633, -181.643, -2143.267]
  MoveL 1117 to (-56.08, 272.6, 260) mm, rotated rx -90 ry -25 rz -52.67 deg; joints [-3.358, -48.759, 103.884, -142.885, 108.641, -181.914, -2147.333]
  MoveL 1118 to (-57.08, 269.15, 270) mm, rotated rx -90 ry -25 rz -49.11 deg; joints [-2.992, -48.637, 103.613, -142.672, 108.649, -182.185, -2150.894]
  MoveL 1119 to (-57.77, 266.15, 280) mm, rotated rx -90 ry -25 rz -46.08 deg; joints [-2.628, -48.509, 103.335, -142.461, 108.657, -182.456, -2153.924]
  MoveL 1120 to (-58.22, 263.67, 290) mm, rotated rx -90 ry -25 rz -43.61 deg; joints [-2.265, -48.376, 103.052, -142.252, 108.666, -182.728, -2156.394]
  Set speed (1000.0 mm/s)
  MoveL 1121 to (-58.22, 263.67, 290) mm, rotated rx -90 ry -25 rz -43.61 deg; joints [-2.265, -48.376, 103.052, -142.252, 108.666, -182.728, -2156.394]
  Set speed (1000.0 mm/s)
  MoveL 1122 to (-78.63, 259.66, 290) mm, rotated rx -90 ry -25 rz -39.75 deg; joints [-2.265, -49.329, 102.952, -142.464, 107.833, -183.405, -2160.245]
  MoveL 1123 to (-78.63, 259.66, 290) mm, rotated rx -90 ry -25 rz -39.75 deg; joints [-2.265, -49.329, 102.952, -142.464, 107.833, -183.405, -2160.245]
  Set speed (60.0 mm/s)
  MoveL 1124 to (-78.34, 263.02, 280) mm, rotated rx -90 ry -25 rz -42.21 deg; joints [-2.628, -49.466, 103.236, -142.672, 107.819, -183.132, -2157.792]
  MoveL 1125 to (-77.78, 267.1, 270) mm, rotated rx -90 ry -25 rz -45.21 deg; joints [-2.992, -49.596, 103.514, -142.883, 107.807, -182.858, -2154.787]
  MoveL 1126 to (-76.86, 271.82, 260) mm, rotated rx -90 ry -25 rz -48.74 deg; joints [-3.358, -49.721, 103.786, -143.095, 107.795, -182.585, -2151.259]
  MoveL 1127 to (-75.48, 277.1, 250) mm, rotated rx -90 ry -25 rz -52.76 deg; joints [-3.725, -49.841, 104.052, -143.309, 107.783, -182.312, -2147.238]
  MoveL 1128 to (-73.51, 282.82, 240) mm, rotated rx -90 ry -25 rz -57.25 deg; joints [-4.093, -49.955, 104.311, -143.526, 107.771, -182.04, -2142.753]
  MoveL 1129 to (-70.88, 288.88, 230) mm, rotated rx -90 ry -25 rz -62.17 deg; joints [-4.463, -50.065, 104.565, -143.744, 107.759, -181.769, -2137.833]
  MoveL 1130 to (-67.49, 295.12, 220) mm, rotated rx -90 ry -25 rz -67.49 deg; joints [-4.834, -50.171, 104.812, -143.964, 107.746, -181.499, -2132.509]
  MoveL 1131 to (-63.28, 301.4, 210) mm, rotated rx -90 ry -25 rz -73.19 deg; joints [-5.207, -50.274, 105.053, -144.186, 107.732, -181.231, -2126.81]
  MoveL 1132 to (-58.22, 307.54, 200) mm, rotated rx -90 ry -25 rz -79.23 deg; joints [-5.581, -50.373, 105.288, -144.411, 107.716, -180.964, -2120.77]
  MoveL 1133 to (-52.31, 313.38, 190) mm, rotated rx -90 ry -25 rz -85.58 deg; joints [-5.956, -50.47, 105.516, -144.637, 107.698, -180.7, -2114.421]
  MoveL 1134 to (-45.56, 318.73, 180) mm, rotated rx -90 ry -25 rz -92.2 deg; joints [-6.332, -50.566, 105.738, -144.867, 107.678, -180.439, -2107.8]
  MoveL 1135 to (-38.04, 323.45, 170) mm, rotated rx -90 ry -25 rz -99.05 deg; joints [-6.709, -50.66, 105.954, -145.098, 107.653, -180.181, -2100.945]
  MoveL 1136 to (-29.85, 327.37, 160) mm, rotated rx -90 ry -25 rz -106.1 deg; joints [-7.088, -50.754, 106.163, -145.333, 107.625, -179.927, -2093.897]
  MoveL 1137 to (-21.11, 330.36, 150) mm, rotated rx -90 ry -25 rz -113.3 deg; joints [-7.468, -50.848, 106.365, -145.57, 107.592, -179.676, -2086.697]
  MoveL 1138 to (-11.96, 332.32, 140) mm, rotated rx -90 ry -25 rz -120.61 deg; joints [-7.849, -50.942, 106.561, -145.81, 107.555, -179.429, -2079.391]
  MoveL 1139 to (-2.59, 333.2, 130) mm, rotated rx -90 ry -25 rz -127.97 deg; joints [-8.231, -51.037, 106.75, -146.052, 107.512, -179.187, -2072.026]
  MoveL 1140 to (6.83, 332.94, 120) mm, rotated rx -90 ry -25 rz -135.35 deg; joints [-8.614, -51.133, 106.932, -146.297, 107.464, -178.949, -2064.647]
  MoveL 1141 to (16.13, 331.57, 110) mm, rotated rx -90 ry -25 rz -142.7 deg; joints [-8.998, -51.23, 107.108, -146.545, 107.41, -178.715, -2057.302]
  MoveL 1142 to (25.11, 329.13, 100) mm, rotated rx -90 ry -25 rz -149.96 deg; joints [-9.383, -51.328, 107.277, -146.795, 107.351, -178.485, -2050.039]
  MoveL 1143 to (33.62, 325.71, 90) mm, rotated rx -90 ry -25 rz -157.1 deg; joints [-9.769, -51.426, 107.439, -147.048, 107.287, -178.259, -2042.902]
  MoveL 1144 to (41.52, 321.41, 80) mm, rotated rx -90 ry -25 rz -164.06 deg; joints [-10.156, -51.524, 107.595, -147.303, 107.218, -178.035, -2035.936]
  MoveL 1145 to (48.7, 316.39, 70) mm, rotated rx -90 ry -25 rz -170.82 deg; joints [-10.544, -51.621, 107.745, -147.56, 107.145, -177.815, -2029.182]
  MoveL 1146 to (55.08, 310.79, 60) mm, rotated rx -90 ry -25 rz -177.32 deg; joints [-10.933, -51.718, 107.888, -147.818, 107.069, -177.598, -2022.679]
  MoveL 1147 to (60.61, 304.79, 50) mm, rotated rx -90 ry -25 rz 176.47 deg; joints [-11.323, -51.812, 108.024, -148.079, 106.99, -177.382, -2016.465]
  MoveL 1148 to (65.29, 298.57, 40) mm, rotated rx -90 ry -25 rz 170.57 deg; joints [-11.713, -51.904, 108.154, -148.341, 106.908, -177.168, -2010.575]
  MoveL 1149 to (69.12, 292.29, 30) mm, rotated rx -90 ry -25 rz 175.04 deg; joints [-12.154, -47.614, 107.647, -146.68, 118.983, -170.079, -2005.041]
  MoveL 1150 to (72.16, 286.11, 20) mm, rotated rx -90 ry -25 rz 169.9 deg; joints [-12.543, -47.695, 107.768, -146.916, 118.909, -169.869, -1999.895]
  MoveL 1151 to (74.48, 280.19, 10) mm, rotated rx -90 ry -25 rz 165.17 deg; joints [-12.934, -47.773, 107.882, -147.153, 118.834, -169.659, -1995.168]
  MoveL 1152 to (76.17, 274.65, 0) mm, rotated rx -90 ry -25 rz 160.89 deg; joints [-13.325, -47.846, 107.991, -147.391, 118.758, -169.451, -1990.889]
  Set speed (1000.0 mm/s)
  MoveL 1153 to (76.17, 274.65, 0) mm, rotated rx -90 ry -25 rz 160.89 deg; joints [-13.325, -47.846, 107.991, -147.391, 118.758, -169.451, -1990.889]
  Set speed (1000.0 mm/s)
  MoveL 1154 to (-78.63, 259.66, 290) mm, rotated rx -90 ry -25 rz -39.75 deg; joints [-2.265, -49.329, 102.952, -142.464, 107.833, -183.405, -2160.245]
  MoveL 1155 to (-78.63, 259.66, 290) mm, rotated rx -90 ry -25 rz -39.75 deg; joints [-2.265, -49.329, 102.952, -142.464, 107.833, -183.405, -2160.245]
  Set speed (60.0 mm/s)
  MoveL 1156 to (-58.93, 252.99, 290) mm, rotated rx -90 ry -25 rz -33.22 deg; joints [-2.265, -48.424, 103.048, -142.262, 108.625, -182.762, -2166.784]
  Set speed (1000.0 mm/s)
  MoveL 1157 to (-58.93, 252.99, 290) mm, rotated rx -90 ry -25 rz -33.22 deg; joints [-2.265, -48.424, 103.048, -142.262, 108.625, -182.762, -2166.784]
  Set speed (1000.0 mm/s)
  MoveL 1158 to (76.17, 274.65, 0) mm, rotated rx -90 ry -25 rz 160.89 deg; joints [-13.325, -47.846, 107.991, -147.391, 118.758, -169.451, -1990.889]
  MoveL 1159 to (76.17, 274.65, 0) mm, rotated rx -90 ry -25 rz 160.89 deg; joints [-13.325, -47.846, 107.991, -147.391, 118.758, -169.451, -1990.889]
  Set speed (60.0 mm/s)
  MoveL 1160 to (55.37, 274.67, 0) mm, rotated rx -90 ry -25 rz 154.84 deg; joints [-13.282, -51.226, 108.712, -149.23, 107.521, -175.73, -1994.838]
  Set speed (1000.0 mm/s)
  MoveL 1161 to (55.37, 274.67, 0) mm, rotated rx -90 ry -25 rz 154.84 deg; joints [-13.282, -51.226, 108.712, -149.23, 107.521, -175.73, -1994.838]
  Set speed (1000.0 mm/s)
  MoveL 1162 to (76.17, 274.65, 0) mm, rotated rx -90 ry -25 rz 160.89 deg; joints [-13.325, -47.846, 107.991, -147.391, 118.758, -169.451, -1990.889]
  MoveL 1163 to (76.17, 274.65, 0) mm, rotated rx -90 ry -25 rz 160.89 deg; joints [-13.325, -47.846, 107.991, -147.391, 118.758, -169.451, -1990.889]
  Set speed (60.0 mm/s)
  MoveL 1164 to (74.48, 280.19, 10) mm, rotated rx -90 ry -25 rz 165.17 deg; joints [-12.934, -47.773, 107.882, -147.153, 118.834, -169.659, -1995.168]
  MoveL 1165 to (72.16, 286.11, 20) mm, rotated rx -90 ry -25 rz 169.9 deg; joints [-12.543, -47.695, 107.768, -146.916, 118.909, -169.869, -1999.895]
  MoveL 1166 to (69.12, 292.29, 30) mm, rotated rx -90 ry -25 rz 175.04 deg; joints [-12.154, -47.614, 107.647, -146.68, 118.983, -170.079, -2005.041]
  MoveL 1167 to (65.29, 298.57, 40) mm, rotated rx -90 ry -25 rz 170.57 deg; joints [-11.713, -51.904, 108.154, -148.341, 106.908, -177.168, -2010.575]
  MoveL 1168 to (60.61, 304.79, 50) mm, rotated rx -90 ry -25 rz 176.47 deg; joints [-11.323, -51.812, 108.024, -148.079, 106.99, -177.382, -2016.465]
  MoveL 1169 to (55.08, 310.79, 60) mm, rotated rx -90 ry -25 rz -177.32 deg; joints [-10.933, -51.718, 107.888, -147.818, 107.069, -177.598, -2022.679]
  MoveL 1170 to (48.7, 316.39, 70) mm, rotated rx -90 ry -25 rz -170.82 deg; joints [-10.544, -51.621, 107.745, -147.56, 107.145, -177.815, -2029.182]
  MoveL 1171 to (41.52, 321.41, 80) mm, rotated rx -90 ry -25 rz -164.06 deg; joints [-10.156, -51.524, 107.595, -147.303, 107.218, -178.035, -2035.936]
  MoveL 1172 to (33.62, 325.71, 90) mm, rotated rx -90 ry -25 rz -157.1 deg; joints [-9.769, -51.426, 107.439, -147.048, 107.287, -178.259, -2042.902]
  MoveL 1173 to (25.11, 329.13, 100) mm, rotated rx -90 ry -25 rz -149.96 deg; joints [-9.383, -51.328, 107.277, -146.795, 107.351, -178.485, -2050.039]
  MoveL 1174 to (16.13, 331.57, 110) mm, rotated rx -90 ry -25 rz -142.7 deg; joints [-8.998, -51.23, 107.108, -146.545, 107.41, -178.715, -2057.302]
  MoveL 1175 to (6.83, 332.94, 120) mm, rotated rx -90 ry -25 rz -135.35 deg; joints [-8.614, -51.133, 106.932, -146.297, 107.464, -178.949, -2064.647]
  MoveL 1176 to (-2.59, 333.2, 130) mm, rotated rx -90 ry -25 rz -127.97 deg; joints [-8.231, -51.037, 106.75, -146.052, 107.512, -179.187, -2072.026]
  MoveL 1177 to (-11.96, 332.32, 140) mm, rotated rx -90 ry -25 rz -120.61 deg; joints [-7.849, -50.942, 106.561, -145.81, 107.555, -179.429, -2079.391]
  MoveL 1178 to (-21.11, 330.36, 150) mm, rotated rx -90 ry -25 rz -113.3 deg; joints [-7.468, -50.848, 106.365, -145.57, 107.592, -179.676, -2086.697]
  MoveL 1179 to (-29.85, 327.37, 160) mm, rotated rx -90 ry -25 rz -106.1 deg; joints [-7.088, -50.754, 106.163, -145.333, 107.625, -179.927, -2093.897]
  MoveL 1180 to (-38.04, 323.45, 170) mm, rotated rx -90 ry -25 rz -99.05 deg; joints [-6.709, -50.66, 105.954, -145.098, 107.653, -180.181, -2100.945]
  MoveL 1181 to (-45.56, 318.73, 180) mm, rotated rx -90 ry -25 rz -92.2 deg; joints [-6.332, -50.566, 105.738, -144.867, 107.678, -180.439, -2107.8]
  MoveL 1182 to (-52.31, 313.38, 190) mm, rotated rx -90 ry -25 rz -85.58 deg; joints [-5.956, -50.47, 105.516, -144.637, 107.698, -180.7, -2114.421]
  MoveL 1183 to (-58.22, 307.54, 200) mm, rotated rx -90 ry -25 rz -79.23 deg; joints [-5.581, -50.373, 105.288, -144.411, 107.716, -180.964, -2120.77]
  MoveL 1184 to (-63.28, 301.4, 210) mm, rotated rx -90 ry -25 rz -73.19 deg; joints [-5.207, -50.274, 105.053, -144.186, 107.732, -181.231, -2126.81]
  MoveL 1185 to (-67.49, 295.12, 220) mm, rotated rx -90 ry -25 rz -67.49 deg; joints [-4.834, -50.171, 104.812, -143.964, 107.746, -181.499, -2132.509]
  MoveL 1186 to (-70.88, 288.88, 230) mm, rotated rx -90 ry -25 rz -62.17 deg; joints [-4.463, -50.065, 104.565, -143.744, 107.759, -181.769, -2137.833]
  MoveL 1187 to (-73.51, 282.82, 240) mm, rotated rx -90 ry -25 rz -57.25 deg; joints [-4.093, -49.955, 104.311, -143.526, 107.771, -182.04, -2142.753]
  MoveL 1188 to (-75.48, 277.1, 250) mm, rotated rx -90 ry -25 rz -52.76 deg; joints [-3.725, -49.841, 104.052, -143.309, 107.783, -182.312, -2147.238]
  MoveL 1189 to (-76.86, 271.82, 260) mm, rotated rx -90 ry -25 rz -48.74 deg; joints [-3.358, -49.721, 103.786, -143.095, 107.795, -182.585, -2151.259]
  MoveL 1190 to (-77.78, 267.1, 270) mm, rotated rx -90 ry -25 rz -45.21 deg; joints [-2.992, -49.596, 103.514, -142.883, 107.807, -182.858, -2154.787]
  MoveL 1191 to (-78.34, 263.02, 280) mm, rotated rx -90 ry -25 rz -42.21 deg; joints [-2.628, -49.466, 103.236, -142.672, 107.819, -183.132, -2157.792]
  MoveL 1192 to (-78.63, 259.66, 290) mm, rotated rx -90 ry -25 rz -39.75 deg; joints [-2.265, -49.329, 102.952, -142.464, 107.833, -183.405, -2160.245]
  Set speed (1000.0 mm/s)
  MoveL 1193 to (-78.63, 259.66, 290) mm, rotated rx -90 ry -25 rz -39.75 deg; joints [-2.265, -49.329, 102.952, -142.464, 107.833, -183.405, -2160.245]
  Set speed (1000.0 mm/s)
  MoveL 1194 to (-58.93, 252.99, 290) mm, rotated rx -90 ry -25 rz -33.22 deg; joints [-2.265, -48.424, 103.048, -142.262, 108.625, -182.762, -2166.784]
  MoveL 1195 to (-58.93, 252.99, 290) mm, rotated rx -90 ry -25 rz -33.22 deg; joints [-2.265, -48.424, 103.048, -142.262, 108.625, -182.762, -2166.784]
  Set speed (60.0 mm/s)
  MoveL 1196 to (-58.94, 255.51, 280) mm, rotated rx -90 ry -25 rz -35.64 deg; joints [-2.628, -48.557, 103.331, -142.472, 108.616, -182.49, -2164.356]
  MoveL 1197 to (-58.8, 258.59, 270) mm, rotated rx -90 ry -25 rz -38.62 deg; joints [-2.992, -48.685, 103.608, -142.683, 108.607, -182.218, -2161.378]
  MoveL 1198 to (-58.44, 262.16, 260) mm, rotated rx -90 ry -25 rz -42.12 deg; joints [-3.358, -48.807, 103.88, -142.896, 108.599, -181.947, -2157.879]
  MoveL 1199 to (-57.77, 266.19, 250) mm, rotated rx -90 ry -25 rz -46.12 deg; joints [-3.725, -48.924, 104.145, -143.111, 108.592, -181.676, -2153.884]
  MoveL 1200 to (-56.69, 270.59, 240) mm, rotated rx -90 ry -25 rz -50.58 deg; joints [-4.093, -49.035, 104.404, -143.327, 108.584, -181.405, -2149.42]
  MoveL 1201 to (-55.14, 275.28, 230) mm, rotated rx -90 ry -25 rz -55.49 deg; joints [-4.463, -49.142, 104.657, -143.546, 108.577, -181.135, -2144.512]
  MoveL 1202 to (-53.04, 280.16, 220) mm, rotated rx -90 ry -25 rz -60.81 deg; joints [-4.834, -49.244, 104.904, -143.767, 108.569, -180.867, -2139.189]
  MoveL 1203 to (-50.33, 285.12, 210) mm, rotated rx -90 ry -25 rz -66.52 deg; joints [-5.207, -49.343, 105.144, -143.99, 108.56, -180.6, -2133.477]
  MoveL 1204 to (-46.98, 290.04, 200) mm, rotated rx -90 ry -25 rz -72.6 deg; joints [-5.581, -49.438, 105.378, -144.215, 108.549, -180.335, -2127.405]
  MoveL 1205 to (-42.97, 294.79, 190) mm, rotated rx -90 ry -25 rz -79 deg; joints [-5.956, -49.531, 105.606, -144.442, 108.537, -180.072, -2121.005]
  MoveL 1206 to (-38.31, 299.24, 180) mm, rotated rx -90 ry -25 rz -85.69 deg; joints [-6.332, -49.621, 105.828, -144.672, 108.522, -179.811, -2114.31]
  MoveL 1207 to (-33.03, 303.26, 170) mm, rotated rx -90 ry -25 rz -92.64 deg; joints [-6.709, -49.71, 106.043, -144.904, 108.504, -179.554, -2107.357]
  MoveL 1208 to (-27.19, 306.74, 160) mm, rotated rx -90 ry -25 rz -99.81 deg; joints [-7.088, -49.799, 106.252, -145.139, 108.483, -179.301, -2100.187]
  MoveL 1209 to (-20.88, 309.56, 150) mm, rotated rx -90 ry -25 rz -107.16 deg; joints [-7.468, -49.887, 106.454, -145.376, 108.457, -179.051, -2092.844]
  MoveL 1210 to (-14.2, 311.65, 140) mm, rotated rx -90 ry -25 rz -114.63 deg; joints [-7.849, -49.976, 106.65, -145.617, 108.426, -178.805, -2085.374]
  MoveL 1211 to (-7.28, 312.93, 130) mm, rotated rx -90 ry -25 rz -122.17 deg; joints [-8.231, -50.066, 106.839, -145.86, 108.39, -178.563, -2077.828]
  MoveL 1212 to (-0.24, 313.38, 120) mm, rotated rx -90 ry -25 rz -129.74 deg; joints [-8.614, -50.157, 107.022, -146.106, 108.349, -178.326, -2070.258]
  MoveL 1213 to (6.77, 312.99, 110) mm, rotated rx -90 ry -25 rz -137.29 deg; joints [-8.998, -50.249, 107.198, -146.354, 108.302, -178.093, -2062.715]
  MoveL 1214 to (13.63, 311.79, 100) mm, rotated rx -90 ry -25 rz -144.75 deg; joints [-9.383, -50.343, 107.367, -146.605, 108.25, -177.865, -2055.252]
  MoveL 1215 to (20.21, 309.81, 90) mm, rotated rx -90 ry -25 rz -152.08 deg; joints [-9.769, -50.437, 107.531, -146.859, 108.193, -177.64, -2047.921]
  MoveL 1216 to (26.38, 307.15, 80) mm, rotated rx -90 ry -25 rz -159.23 deg; joints [-10.156, -50.531, 107.687, -147.115, 108.13, -177.419, -2040.769]
  MoveL 1217 to (32.08, 303.89, 70) mm, rotated rx -90 ry -25 rz -166.16 deg; joints [-10.544, -50.625, 107.837, -147.374, 108.064, -177.201, -2033.843]
  MoveL 1218 to (37.21, 300.16, 60) mm, rotated rx -90 ry -25 rz -172.82 deg; joints [-10.933, -50.719, 107.981, -147.634, 107.993, -176.986, -2027.185]
  MoveL 1219 to (41.73, 296.07, 50) mm, rotated rx -90 ry -25 rz -179.17 deg; joints [-11.323, -50.811, 108.119, -147.896, 107.919, -176.773, -2020.833]
  MoveL 1220 to (45.64, 291.75, 40) mm, rotated rx -90 ry -25 rz 174.82 deg; joints [-11.713, -50.9, 108.25, -148.16, 107.843, -176.562, -2014.824]
  MoveL 1221 to (48.92, 287.33, 30) mm, rotated rx -90 ry -25 rz 169.19 deg; joints [-12.104, -50.987, 108.375, -148.426, 107.764, -176.353, -2009.19]
  MoveL 1222 to (51.6, 282.93, 20) mm, rotated rx -90 ry -25 rz 163.96 deg; joints [-12.496, -51.071, 108.493, -148.693, 107.684, -176.144, -2003.962]
  MoveL 1223 to (53.73, 278.68, 10) mm, rotated rx -90 ry -25 rz 159.17 deg; joints [-12.889, -51.151, 108.606, -148.961, 107.602, -175.937, -1999.169]
  MoveL 1224 to (55.37, 274.67, 0) mm, rotated rx -90 ry -25 rz 154.84 deg; joints [-13.282, -51.226, 108.712, -149.23, 107.521, -175.73, -1994.838]
  Set speed (1000.0 mm/s)
  MoveL 1225 to (55.37, 274.67, 0) mm, rotated rx -90 ry -25 rz 154.84 deg; joints [-13.282, -51.226, 108.712, -149.23, 107.521, -175.73, -1994.838]
  Set speed (1000.0 mm/s)
  MoveL 1226 to (-58.93, 252.99, 290) mm, rotated rx -90 ry -25 rz -33.22 deg; joints [-2.265, -48.424, 103.048, -142.262, 108.625, -182.762, -2166.784]
  MoveL 1227 to (-58.93, 252.99, 290) mm, rotated rx -90 ry -25 rz -33.22 deg; joints [-2.265, -48.424, 103.048, -142.262, 108.625, -182.762, -2166.784]
  Set speed (60.0 mm/s)
  MoveL 1228 to (-37.11, 208.63, 290) mm, rotated rx -90 ry -25 rz 14.16 deg; joints [-2.265, -48.614, 103.03, -142.305, 108.461, -182.896, -2214.156]
  Set speed (1000.0 mm/s)
  MoveL 1229 to (-37.11, 208.63, 290) mm, rotated rx -90 ry -25 rz 14.16 deg; joints [-2.265, -48.614, 103.03, -142.305, 108.461, -182.896, -2214.156]
  Set speed (1000.0 mm/s)
  MoveL 1230 to (55.37, 274.67, 0) mm, rotated rx -90 ry -25 rz 154.84 deg; joints [-13.282, -51.226, 108.712, -149.23, 107.521, -175.73, -2354.838]
  MoveL 1231 to (55.37, 274.67, 0) mm, rotated rx -90 ry -25 rz 154.84 deg; joints [-13.282, -51.226, 108.712, -149.23, 107.521, -175.73, -2354.838]
  Set speed (60.0 mm/s)
  MoveL 1232 to (20.49, 309.71, 0) mm, rotated rx -90 ry -25 rz -152.4 deg; joints [-13.282, -51.049, 108.726, -149.199, 107.684, -175.627, -2407.595]
  Set speed (1000.0 mm/s)
  MoveL 1233 to (20.49, 309.71, 0) mm, rotated rx -90 ry -25 rz -152.4 deg; joints [-13.282, -51.049, 108.726, -149.199, 107.684, -175.627, -2407.595]
  Set speed (1000.0 mm/s)
  MoveL 1234 to (55.37, 274.67, 0) mm, rotated rx -90 ry -25 rz 154.84 deg; joints [-13.282, -51.226, 108.712, -149.23, 107.521, -175.73, -2354.838]
  MoveL 1235 to (55.37, 274.67, 0) mm, rotated rx -90 ry -25 rz 154.84 deg; joints [-13.282, -51.226, 108.712, -149.23, 107.521, -175.73, -2354.838]
  Set speed (60.0 mm/s)
  MoveL 1236 to (53.73, 278.68, 10) mm, rotated rx -90 ry -25 rz 159.17 deg; joints [-12.889, -51.151, 108.606, -148.961, 107.602, -175.937, -2359.169]
  MoveL 1237 to (51.6, 282.93, 20) mm, rotated rx -90 ry -25 rz 163.96 deg; joints [-12.496, -51.071, 108.493, -148.693, 107.684, -176.144, -2363.962]
  MoveL 1238 to (48.92, 287.33, 30) mm, rotated rx -90 ry -25 rz 169.19 deg; joints [-12.104, -50.987, 108.375, -148.426, 107.764, -176.353, -2369.19]
  MoveL 1239 to (45.64, 291.75, 40) mm, rotated rx -90 ry -25 rz 174.82 deg; joints [-11.713, -50.9, 108.25, -148.16, 107.843, -176.562, -2374.824]
  MoveL 1240 to (41.73, 296.07, 50) mm, rotated rx -90 ry -25 rz -179.17 deg; joints [-11.323, -50.811, 108.119, -147.896, 107.919, -176.773, -2380.833]
  MoveL 1241 to (37.21, 300.16, 60) mm, rotated rx -90 ry -25 rz -172.82 deg; joints [-10.933, -50.719, 107.981, -147.634, 107.993, -176.986, -2387.185]
  MoveL 1242 to (32.08, 303.89, 70) mm, rotated rx -90 ry -25 rz -166.16 deg; joints [-10.544, -50.625, 107.837, -147.374, 108.064, -177.201, -2393.843]
  MoveL 1243 to (26.38, 307.15, 80) mm, rotated rx -90 ry -25 rz -159.23 deg; joints [-10.156, -50.531, 107.687, -147.115, 108.13, -177.419, -2400.769]
  MoveL 1244 to (20.21, 309.81, 90) mm, rotated rx -90 ry -25 rz -152.08 deg; joints [-9.769, -50.437, 107.531, -146.859, 108.193, -177.64, -2407.921]
  MoveL 1245 to (13.63, 311.79, 100) mm, rotated rx -90 ry -25 rz -144.75 deg; joints [-9.383, -50.343, 107.367, -146.605, 108.25, -177.865, -2415.252]
  MoveL 1246 to (6.77, 312.99, 110) mm, rotated rx -90 ry -25 rz -137.29 deg; joints [-8.998, -50.249, 107.198, -146.354, 108.302, -178.093, -2422.715]
  MoveL 1247 to (-0.24, 313.38, 120) mm, rotated rx -90 ry -25 rz -129.74 deg; joints [-8.614, -50.157, 107.022, -146.106, 108.349, -178.326, -2430.258]
  MoveL 1248 to (-7.28, 312.93, 130) mm, rotated rx -90 ry -25 rz -122.17 deg; joints [-8.231, -50.066, 106.839, -145.86, 108.39, -178.563, -2437.828]
  MoveL 1249 to (-14.2, 311.65, 140) mm, rotated rx -90 ry -25 rz -114.63 deg; joints [-7.849, -49.976, 106.65, -145.617, 108.426, -178.805, -2445.374]
  MoveL 1250 to (-20.88, 309.56, 150) mm, rotated rx -90 ry -25 rz -107.16 deg; joints [-7.468, -49.887, 106.454, -145.376, 108.457, -179.051, -2452.844]
  MoveL 1251 to (-27.19, 306.74, 160) mm, rotated rx -90 ry -25 rz -99.81 deg; joints [-7.088, -49.799, 106.252, -145.139, 108.483, -179.301, -2460.187]
  MoveL 1252 to (-33.03, 303.26, 170) mm, rotated rx -90 ry -25 rz -92.64 deg; joints [-6.709, -49.71, 106.043, -144.904, 108.504, -179.554, -2467.357]
  MoveL 1253 to (-38.31, 299.24, 180) mm, rotated rx -90 ry -25 rz -85.69 deg; joints [-6.332, -49.621, 105.828, -144.672, 108.522, -179.811, -2474.31]
  MoveL 1254 to (-42.97, 294.79, 190) mm, rotated rx -90 ry -25 rz -79 deg; joints [-5.956, -49.531, 105.606, -144.442, 108.537, -180.072, -2481.005]
  MoveL 1255 to (-46.98, 290.04, 200) mm, rotated rx -90 ry -25 rz -72.6 deg; joints [-5.581, -49.438, 105.378, -144.215, 108.549, -180.335, -2487.405]
  MoveL 1256 to (-50.33, 285.12, 210) mm, rotated rx -90 ry -25 rz -66.52 deg; joints [-5.207, -49.343, 105.144, -143.99, 108.56, -180.6, -2493.477]
  MoveL 1257 to (-53.04, 280.16, 220) mm, rotated rx -90 ry -25 rz -60.81 deg; joints [-4.834, -49.244, 104.904, -143.767, 108.569, -180.867, -2499.189]
  MoveL 1258 to (-55.14, 275.28, 230) mm, rotated rx -90 ry -25 rz -55.49 deg; joints [-4.463, -49.142, 104.657, -143.546, 108.577, -181.135, -2504.512]
  MoveL 1259 to (-56.69, 270.59, 240) mm, rotated rx -90 ry -25 rz -50.58 deg; joints [-4.093, -49.035, 104.404, -143.327, 108.584, -181.405, -2509.42]
  MoveL 1260 to (-57.77, 266.19, 250) mm, rotated rx -90 ry -25 rz -46.12 deg; joints [-3.725, -48.924, 104.145, -143.111, 108.592, -181.676, -2513.884]
  MoveL 1261 to (-58.44, 262.16, 260) mm, rotated rx -90 ry -25 rz -42.12 deg; joints [-3.358, -48.807, 103.88, -142.896, 108.599, -181.947, -2517.879]
  MoveL 1262 to (-58.8, 258.59, 270) mm, rotated rx -90 ry -25 rz -38.62 deg; joints [-2.992, -48.685, 103.608, -142.683, 108.607, -182.218, -2521.378]
  MoveL 1263 to (-58.94, 255.51, 280) mm, rotated rx -90 ry -25 rz -35.64 deg; joints [-2.628, -48.557, 103.331, -142.472, 108.616, -182.49, -2524.356]
  MoveL 1264 to (-58.93, 252.99, 290) mm, rotated rx -90 ry -25 rz -33.22 deg; joints [-2.265, -48.424, 103.048, -142.262, 108.625, -182.762, -2526.784]
  Set speed (1000.0 mm/s)
  MoveL 1265 to (-58.93, 252.99, 290) mm, rotated rx -90 ry -25 rz -33.22 deg; joints [-2.265, -48.424, 103.048, -142.262, 108.625, -182.762, -2526.784]
  Set speed (1000.0 mm/s)
  MoveL 1266 to (-37.11, 208.63, 290) mm, rotated rx -90 ry -25 rz 14.16 deg; joints [-2.265, -48.614, 103.03, -142.305, 108.461, -182.896, -2574.156]
  MoveL 1267 to (-37.11, 208.63, 290) mm, rotated rx -90 ry -25 rz 14.16 deg; joints [-2.265, -48.614, 103.03, -142.305, 108.461, -182.896, -2574.156]
  Set speed (60.0 mm/s)
  MoveL 1268 to (-39.03, 210.26, 280) mm, rotated rx -90 ry -25 rz 11.88 deg; joints [-2.628, -48.753, 103.313, -142.515, 108.447, -182.627, -2571.877]
  MoveL 1269 to (-41.29, 212.35, 270) mm, rotated rx -90 ry -25 rz 9.09 deg; joints [-2.992, -48.886, 103.59, -142.727, 108.433, -182.358, -2569.089]
  MoveL 1270 to (-43.78, 214.95, 260) mm, rotated rx -90 ry -25 rz 5.82 deg; joints [-3.358, -49.014, 103.861, -142.941, 108.42, -182.09, -2565.82]
